// TIA Portal V20 export
// export: Created 2025-12-01T14:57:39.3017636Z, ExportSetting None, DisplayName Totally Integrated Automation Portal, DisplayVersion V20 Update 3, DisplayName TIA Portal Openness, DisplayVersion V20 Update 3, DisplayName TIA Portal Version Control Interface, DisplayVersion V20 Update 3, DisplayName STEP 7 Professional, DisplayVersion V20 Update 3, DisplayName STEP 7 Safety, DisplayVersion V20 Update 2, DisplayName WinCC Basic/Comfort/Advanced, DisplayVersion V20 Update 3, DisplayName WinCC Professional, DisplayVersion V20 Update 3, DisplayName WinCC Unified, DisplayVersion V20 Update 3
FUNCTION_BLOCK "FB370_ApiladorDeCajasPlastico"   // FB370, LAD
TITLE = Apilador de Cajas de Plastico
{ S7_Optimized_Access := 'FALSE' }
AUTHOR : MAQUINA
NAME : 20160211
VERSION : 3.2
// Dani Palacios: Modificación octubre 2017 para poder desabilitar la maquina con un bit (por ejemplo en la puesta a punto si no esta montada o en el simulador)
// La modificación esta sin probar y es todo lo relativo a la variable Maquina_Desabilitada
// (bloqueo evolución desde etapa 0, bloqueo activación salidas en etapa 0 , fin vi sin mirar detectores y activación posición de reposo sin mirar detectores y variabkles de fin de movimiento).
// ES RESPONSABILIDAD DEL QUE DESABILITA LA MAQUINA QUE ESTA ESTE EN UNA POSICION QUE PERMITA EL MOVIMIENTO DE LAS CARGAS A TRAVES DE ELLA
// stored: AutoNumber false, SetENOAutomatically false
   VAR_INPUT
      Maquina : UInt;   // Numero de Maquina (Mesa)
      Error_Tx : Bool;   // Error en el Tx
      EnTension : Bool;   // Existe Tension en la Mesa
      NodoNoPresente : Bool;   // Nodo No Presente >>> Var. LENZE de Elevacion
      ByteInicial : Int;   // Byte Inicial >>> Var. LENZE de Elevacion
      MAQx_DesHabilitada : Bool;   // Config MAQ. >>> DesHabilitada
      MAQx_SinPrimerCentrado : Bool;   // Config MAQ. >>> No Activar Primer Centrado (Antes de Entrada)
      MAQx_ActivarEspera : Bool;   // Config MAQ. >>> Sin Espera en Etapas
      MAQx_SinTopes : Bool;   // Config MAQ. >>> Sin Utilizar Topes (Los Centradores)
      TermicoFreno_ELEV : Bool;   // Termico del Freno de la Elevacion
      pHsMx_PresCarga : Bool;   // pHs de Presencia de Carga en la Maquina
      pHsMx_1 : Bool;   // pHs de la Mesa - Pos 1 de Av
      pHsMx_2 : Bool;   // pHs de la Mesa - Pos 2 de Av
      pHsMx_CtrEntrada : Bool;   // pHs Control de Entrada de Seguridad
      pHs_Referencia : Bool;   // pHs de Referencia >>> Var. LENZE de Elevacion
      EM_Up : Bool;   // Emergencia Arriba >>> Var. LENZE de Elevacion
      EM_Down : Bool;   // Emergencia Abajo >>> Var. LENZE de Elevacion
      CF1CF2_Cerrado : Bool;   // Centradores 1 y 2 Cerrados
      CF3CF4_Cerrado : Bool;   // Centradores 3 y 4 Cerrados
      CF5CF6_Cerrado : Bool;   // Centradores 5 y 6 Cerrados
      CF1CF2_Abierto : Bool;   // Centradores 1 y 2 Abiertos
      CF3CF4_Abierto : Bool;   // Centradores 3 y 4 Abiertos
      CF5CF6_Abierto : Bool;   // Centradores 5 y 6 Abiertos
      CM1CM2_Cerrado : Bool;   // Garras 1 y 2 Cerradas
      CM3CM4_Cerrado : Bool;   // Garras 3 y 4 Cerradas
      CM5CM6_Cerrado : Bool;   // Garras 5 y 6 Cerradas
      CM7CM8_Cerrado : Bool;   // Garras 7 y 8 Cerradas
      CM9CM10_Cerrado : Bool;   // Garras 9 y 10 Cerradas
      CM1CM2_Abierto : Bool;   // Garras 1 y 2 Abiertas
      CM3CM4_Abierto : Bool;   // Garras 3 y 4 Abiertas
      CM5CM6_Abierto : Bool;   // Garras 5 y 6 Abiertas
      CM7CM8_Abierto : Bool;   // Garras 7 y 8 Abiertas
      CM9CM10_Abierto : Bool;   // Garras 9 y 10 Abiertas
      GF1GF2_Cerrado : Bool;   // Guias superiores 1 y 2 Cerradas
      GF3GF4_Cerrado : Bool;   // Guias superiores 3 y 4 Cerradas
      GF1GF2_Abierto : Bool;   // Guias superiores 1 y 2 Abiertas
      GF3GF4_Abierto : Bool;   // Guias superiores 3 y 4 Abiertas
      EnMov_Centradores : Bool;   // Centradores >>> En Movimiento
      EnMov_Garras : Bool;   // Garras >>> En Movimiento
      EnMov_Guias : Bool;   // Guias >>> En Movimiento
      EnMov_Topes : Bool;   // Topes >>> En Movimiento
      SubirManual : Bool;   // Subir en Manual >>> Var. LENZE de Elevacion
      BajarManual : Bool;   // Bajar en Manual >>> Var. LENZE de Elevacion
      AutoManual : Bool;   // Posicionar en Manual (Para realizar Test de Posicion)
      Homing : Bool;   // Homing >>> Var. LENZE de Elevacion
      CajaGrande_EnEntrada : Bool;   // Caja Grande en Entrada >>> Interlock Mesa
      Apilador_AvisoEntrada : Bool;   // Aviso Entrada >>> Interlock Mesa
      Apilador_FinEntrada : Bool;   // FIn Entrada >>> Interlock Mesa
      ActivarGuias : Bool;   // Activar las Guias Superiores (Por altura de la Pila)
      V_TOut_MovVertical : Int := 15000;   // TimeOut del Movimiento Vertical
      V_TOut_Centradores : Int := 5000;   // TimeOut de los Centradores
      V_TOut_Garras : Int := 5000;   // TimeOut de las Garras
      V_TOut_Guias : Int := 5000;   // TimeOut de las Guias Superiores
      V_TOut_Topes : Int := 5000;   // TimeOut de los Topes
   END_VAR
   VAR_OUTPUT
      Apilador_EnReposo : Bool;   // En Reposo >>> Interlock Maquina
      Apialdor_PermisoEntrada : Bool;   // Permiso deEntrada >>> Interlock Maquina
   END_VAR
   VAR
      PosicionActual : Int;   // Var. LENZE de Elevacion >>> Posicion Actual
      ErrorSubjet : Word;   // Var LENZE de Elevacion
      ErrorID : Word;   // Var LENZE de Elevacion
      PosicionManual : UInt;   // Posicion para el Test Manual
      PosicionInicial : UInt;   // TRACKING >>> Posicion Inicial de la Orden de DesApilar Cajas
      PosicionFinal : UInt;   // TRACKING >>> Posicion Final de la Orden de DesApilar Cajas
      PosicionPreviaInicial : UInt;   // TRACKING >>> Posicion Previa a la inicial - Adelanto de Movimiento
      TipoAmarre : UInt;   // TRACKING >>> Tipo de Amarre de las Garras de la Orden de DesApilar Cajas
      OrdenApilar : Bool;   // TRACKING >>> Orden de DesApilar Cajas
      Fin_OrdenApilar : Bool;   // TRACKING >>> Fin de la Orden de DesApilar Cajas
      Caja_TipoEuroPool : Bool;   // TRACKING >>> Caja de tipo EuroPool
      Caja_DosPequenas : Bool;   // TRACKING >>> La Fila es de Dos Cajas Pequeñas
      Caja_UnaPequena : Bool;   // TRACKING >>> La Fila es de Una Caja Pequeña
      Caja_Grande : Bool;   // TRACKING >>> La Fila es de Una Caja Grande
      Reset_ET00 : Bool;
      Reset_ET01 : Bool;
      Apil_ET00 : Bool;
      Apil_ET01 : Bool;
      Apil_ET02 : Bool;
      Apil_ET03 : Bool;
      Apil_ET04 : Bool;
      Apil_ET05 : Bool;
      Apil_ET06 : Bool;
      Apil_ET07 : Bool;
      Apil_ET08 : Bool;
      Apil_ET09 : Bool;
      Apil_ET10 : Bool;
      Apil_ET11 : Bool;
      Apil_ET12 : Bool;
      Apil_ET13 : Bool;
      Apil_ET14 : Bool;
      Apil_ET15 : Bool;
      PosicionIntermedia : UInt;
      Posicion_OrdenMover : UInt;   // AUXILIAR >>> Posicion de la Orden a Mover el Elevacion
      OrdenMover : Bool;   // AUXILIAR >>> Orden de Mover el Elevacion
      Fin_OrdenMover : Bool;   // AUXILIAR >>> Orden de Mover el Elevacion
      MemoPosicionOK : Bool;   // AUXILIAR >>> Memoria de Posicion OK
      Carga_PosicionInicial : Bool;   // CARGA >>> Posicion Incial del Apilado de Cajas
      Carga_PosicionIntermedia : Bool;   // CARGA >>> Posicion Intermedia del Apilado de Cajas
      Carga_PosicionFinal : Bool;   // CARGA >>> Posicion Final del Apilado de Cajas
      Carga_PosicionPreviaIncial : Bool;   // CARGA >>> Posicion Previa Inicial del Apilado de Cajas
      Carga_PosicionManual : Bool;   // CARGA >>> Posicion Manual de la Orden de Test
      ErrorVariador : Bool;   // AUXILIAR >>> Error del Variador
      ReferenciaOK : Bool;   // AUXILIAR >>> Referencia OK del Variador
      MemoHomingAuto : Bool;   // AUXILIAR >>> Memoria del Homing Automatico del Variador
      TIM_EsperaMover { S7_SetPoint := 'True'} : TON_TIME;   // TIM de Espera de Activar Orden al Var de LENZE (200ms)
      TIM_EsperaET02 { S7_SetPoint := 'True'} : TON_TIME;   // TIM de Espera para Activar ET02 (100ms)
      TIM_EsperaET05 { S7_SetPoint := 'True'} : TON_TIME;   // TIM de Espera para Activar ET05 (100ms)
      TIM_EsperaET13 { S7_SetPoint := 'True'} : TON_TIME;   // TIM de Espera para Activar ET13 (100ms)
      TMP_EnTension { S7_SetPoint := 'True'} : "FB910_CNT_UHS";
      TOut_MovVertical { S7_SetPoint := 'True'} : "FB910_CNT_UHS";   // TimeOut del Movimiento Vertical
      TOut_Centradores { S7_SetPoint := 'True'} : "FB910_CNT_UHS";   // TimeOut de los Centradores
      TOut_Garras { S7_SetPoint := 'True'} : "FB910_CNT_UHS";   // TimeOut de las Garras
      TOut_Guias { S7_SetPoint := 'True'} : "FB910_CNT_UHS";   // TimeOut de las Guias Superiores
      TOut_Topes { S7_SetPoint := 'True'} : "FB910_CNT_UHS";   // TimeOut de los Topes
      MA_Cerrar_CF1CF2 : Bool;   // ????
      MA_Cerrar_CF3CF4 : Bool;   // ????
      MA_Cerrar_CF5CF6 : Bool;   // ????
      MA_Abrir_CF1CF2 : Bool;   // ????
      MA_Abrir_CF3CF4 : Bool;   // ????
      MA_Abrir_CF5CF6 { ExternalVisible := 'False'} : Bool;   // ????
      MA_Cerrar_CM1CM2 : Bool;   // ????
      MA_Cerrar_CM3CM4 : Bool;   // ????
      MA_Cerrar_CM5CM6 : Bool;   // ????
      MA_Cerrar_CM7CM8 : Bool;   // ????
      MA_Cerrar_CM9CM10 : Bool;   // ????
      MA_Abrir_CM1CM2 : Bool;   // ????
      MA_Abrir_CM3CM4 : Bool;   // ????
      MA_Abrir_CM5CM6 : Bool;   // ????
      MA_Abrir_CM7CM8 : Bool;   // ????
      MA_Abrir_CM9CM10 : Bool;   // ????
      MA_Cerrar_GF1GF2 : Bool;   // ????
      MA_Cerrar_GF3GF4 : Bool;   // ????
      MA_Abrir_GF1GF2 : Bool;   // ????
      MA_Abrir_GF3GF4 : Bool;   // ????
   END_VAR
   VAR_TEMP
      EstadoZona : "EstadoZona";   // Estado de Zona de la Mesa
      EstadoMAQ : "EstadoMaquina_ApiladorDeCajasPlastico";   // Estado del Vehiculo Inteliguente de la Maquina
      MAQx_AutoHoming : Bool;   // Config >>> Var. LENZE con Auto Homing
      MAQx_EncoderIncremental : Bool;   // Config >>> Var. LENZE con Encoder Incremental
      MAQx_ActivarAutoManual : Bool;   // Config >>> Activacion para el Test de posicionamiento manual
      MAQx_SinAbrirTopes : Bool;   // Config MAQ. >>> No Abrir Topes - Despues de Entrada
      MAQx_EntradaSinEspera : Bool;   // Config MAQ. >>> No Esperar el Cerrar Topes - Inicio de Entrada
      CentradoresCerrados : Bool;   // AUXILIAR >>> Cerrados los Centradores
      CentradoresAbiertos : Bool;   // AUXILIAR >>> Abiertos los Centradores
      TopesCerrados : Bool;   // AUXILIAR >>> Cerrados los Topes
      GarrasCerradas : Bool;   // AUXILIAR >>> Cerradas las Garras
      GarrasAbiertas : Bool;   // AUXILIAR >>> Abiertas las Garras
      GuiasCerradas : Bool;   // AUXILIAR >>> Cerradas las Guias Superiores
      GuiasAbiertas : Bool;   // AUXILIAR >>> Abiertas las Guias Superiores
      MA_CerrarCentradores : Bool;   // AUXILIAR >>> Cerrar los Centradores
      MA_AbrirCentradores : Bool;   // AUXILIAR >>> Abrir los Centradores
      MA_CerrarTopes : Bool;   // AUXILIAR >>> Cerrar los Topes
      MA_CerrarGarras : Bool;   // AUXILIAR >>> Cerrar las Garras
      MA_AbrirGarras : Bool;   // AUXILIAR >>> Abrir las Garras
      MA_CerrarGuias : Bool;   // AUXILIAR >>> Cerrar las Guias Superiores
      MA_AbrirGuias : Bool;   // AUXILIAR >>> Abrir las Guias Superiores
      Aux_ET00 : Bool;
   END_VAR
BEGIN

REGION Network 1: Configuraciones Especiales - Config >>> Var. LENZE de Elevacion
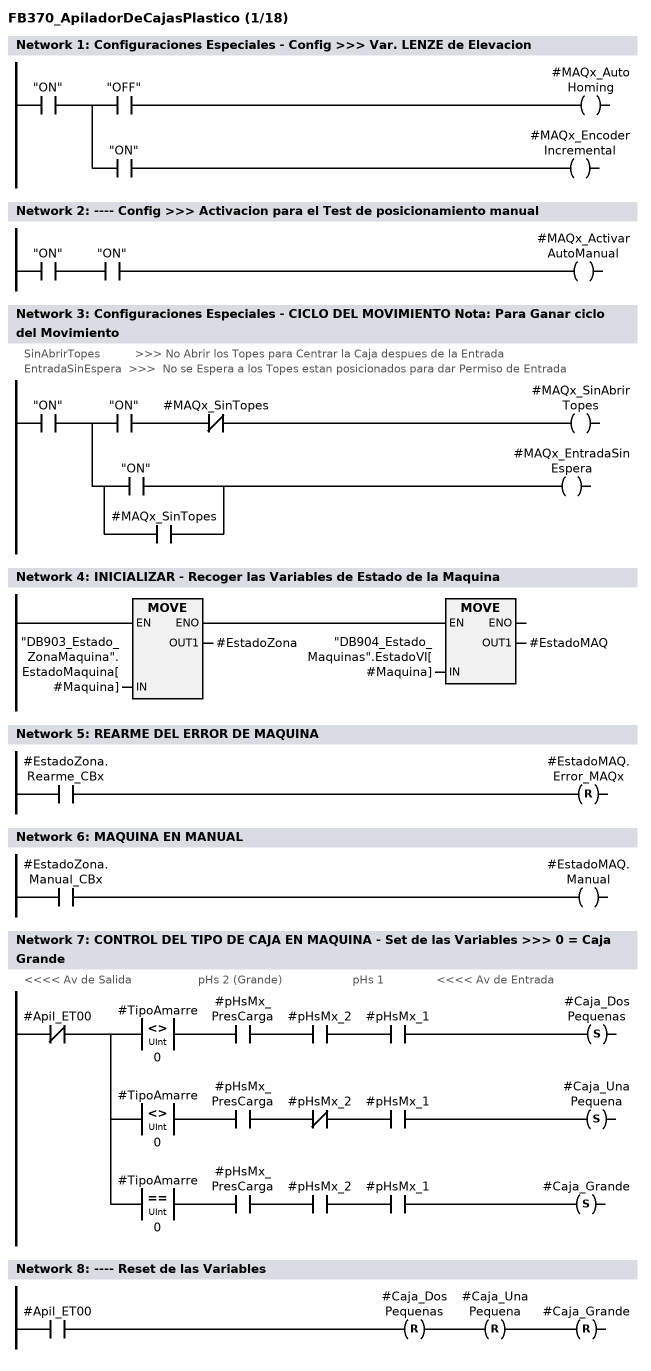
   RUNG wire#powerrail
      Contact( "ON" )
      wire#w1
      Contact( "OFF" )
      Coil( #MAQx_AutoHoming )
   END_RUNG
   RUNG wire#w1
      Contact( "ON" )
      Coil( #MAQx_EncoderIncremental )
   END_RUNG
   // the same network as SCL:
   #MAQx_AutoHoming := "ON" AND "OFF";
   #MAQx_EncoderIncremental := "ON" AND "ON";
END_REGION

REGION Network 2: ---- Config >>> Activacion para el Test de posicionamiento manual
   RUNG wire#powerrail
      Contact( "ON" )
      Contact( "ON" )
      Coil( #MAQx_ActivarAutoManual )
   END_RUNG
   // the same network as SCL:
   #MAQx_ActivarAutoManual := "ON" AND "ON";
END_REGION

REGION Network 3: Configuraciones Especiales - CICLO DEL MOVIMIENTO Nota: Para Ganar ciclo del Movimiento
   // SinAbrirTopes          >>> No Abrir los Topes para Centrar la Caja despues de la Entrada
   // EntradaSinEspera  >>>  No se Espera a los Topes estan posicionados para dar Permiso de Entrada
   RUNG wire#powerrail
      Contact( "ON" )
      wire#w1
      Contact( "ON" )
      I_Contact( #MAQx_SinTopes )
      Coil( #MAQx_SinAbrirTopes )
   END_RUNG
   RUNG wire#w1
      Contact( "ON" )
      wire#w2
      Coil( #MAQx_EntradaSinEspera )
   END_RUNG
   RUNG wire#w1
      Contact( #MAQx_SinTopes )
   END_RUNG wire#w2
   // the same network as SCL:
   #MAQx_SinAbrirTopes := "ON" AND "ON" AND NOT #MAQx_SinTopes;
   #MAQx_EntradaSinEspera := "ON" AND ("ON" OR #MAQx_SinTopes);
END_REGION

REGION Network 4: INICIALIZAR - Recoger las Variables de Estado de la Maquina
   RUNG wire#powerrail
      Move(in := "DB903_Estado_ZonaMaquina".EstadoMaquina[#Maquina], out1 => #EstadoZona)
      Move(in := "DB904_Estado_Maquinas".EstadoVI[#Maquina], out1 => #EstadoMAQ)
   END_RUNG
   // the same network as SCL:
   #EstadoZona := "DB903_Estado_ZonaMaquina".EstadoMaquina[#Maquina];
   #EstadoMAQ := "DB904_Estado_Maquinas".EstadoVI[#Maquina];
END_REGION

REGION Network 5: REARME DEL ERROR DE MAQUINA
   RUNG wire#powerrail
      Contact( #EstadoZona.Rearme_CBx )
      R_Coil( #EstadoMAQ.Error_MAQx )
   END_RUNG
   // the same network as SCL:
   IF #EstadoZona.Rearme_CBx THEN #EstadoMAQ.Error_MAQx := FALSE; END_IF;
END_REGION

REGION Network 6: MAQUINA EN MANUAL
   RUNG wire#powerrail
      Contact( #EstadoZona.Manual_CBx )
      Coil( #EstadoMAQ.Manual )
   END_RUNG
   // the same network as SCL:
   #EstadoMAQ.Manual := #EstadoZona.Manual_CBx;
END_REGION

REGION Network 7: CONTROL DEL TIPO DE CAJA EN MAQUINA - Set de las Variables >>> 0 = Caja Grande
   // <<<< Av de Salida                   pHs 2 (Grande)                    pHs 1               <<<< Av de Entrada
   RUNG wire#powerrail
      I_Contact( #Apil_ET00 )
      wire#w1
      { S7_Templates := "SrcType := UInt" } NE_Contact(in1 := #TipoAmarre, in2 := 0)
      Contact( #pHsMx_PresCarga )
      Contact( #pHsMx_2 )
      Contact( #pHsMx_1 )
      S_Coil( #Caja_DosPequenas )
   END_RUNG
   RUNG wire#w1
      { S7_Templates := "SrcType := UInt" } NE_Contact(in1 := #TipoAmarre, in2 := 0)
      Contact( #pHsMx_PresCarga )
      I_Contact( #pHsMx_2 )
      Contact( #pHsMx_1 )
      S_Coil( #Caja_UnaPequena )
   END_RUNG
   RUNG wire#w1
      { S7_Templates := "SrcType := UInt" } EQ_Contact(in1 := #TipoAmarre, in2 := 0)
      Contact( #pHsMx_PresCarga )
      Contact( #pHsMx_2 )
      Contact( #pHsMx_1 )
      S_Coil( #Caja_Grande )
   END_RUNG
   // the same network as SCL:
   IF NOT #Apil_ET00 AND (#TipoAmarre <> 0) AND #pHsMx_PresCarga AND #pHsMx_2 AND #pHsMx_1 THEN
       #Caja_DosPequenas := TRUE;
   END_IF;
   IF NOT #Apil_ET00 AND (#TipoAmarre <> 0) AND #pHsMx_PresCarga AND NOT #pHsMx_2 AND #pHsMx_1 THEN
       #Caja_UnaPequena := TRUE;
   END_IF;
   IF NOT #Apil_ET00 AND (#TipoAmarre = 0) AND #pHsMx_PresCarga AND #pHsMx_2 AND #pHsMx_1 THEN
       #Caja_Grande := TRUE;
   END_IF;
END_REGION

REGION Network 8: ---- Reset de las Variables
   RUNG wire#powerrail
      Contact( #Apil_ET00 )
      R_Coil( #Caja_DosPequenas )
      R_Coil( #Caja_UnaPequena )
      R_Coil( #Caja_Grande )
   END_RUNG
   // the same network as SCL:
   IF #Apil_ET00 THEN
       #Caja_DosPequenas := FALSE;
       #Caja_UnaPequena := FALSE;
       #Caja_Grande := FALSE;
   END_IF;
END_REGION

REGION Network 9: ---- Config >>> Caja de tipo EuroPool
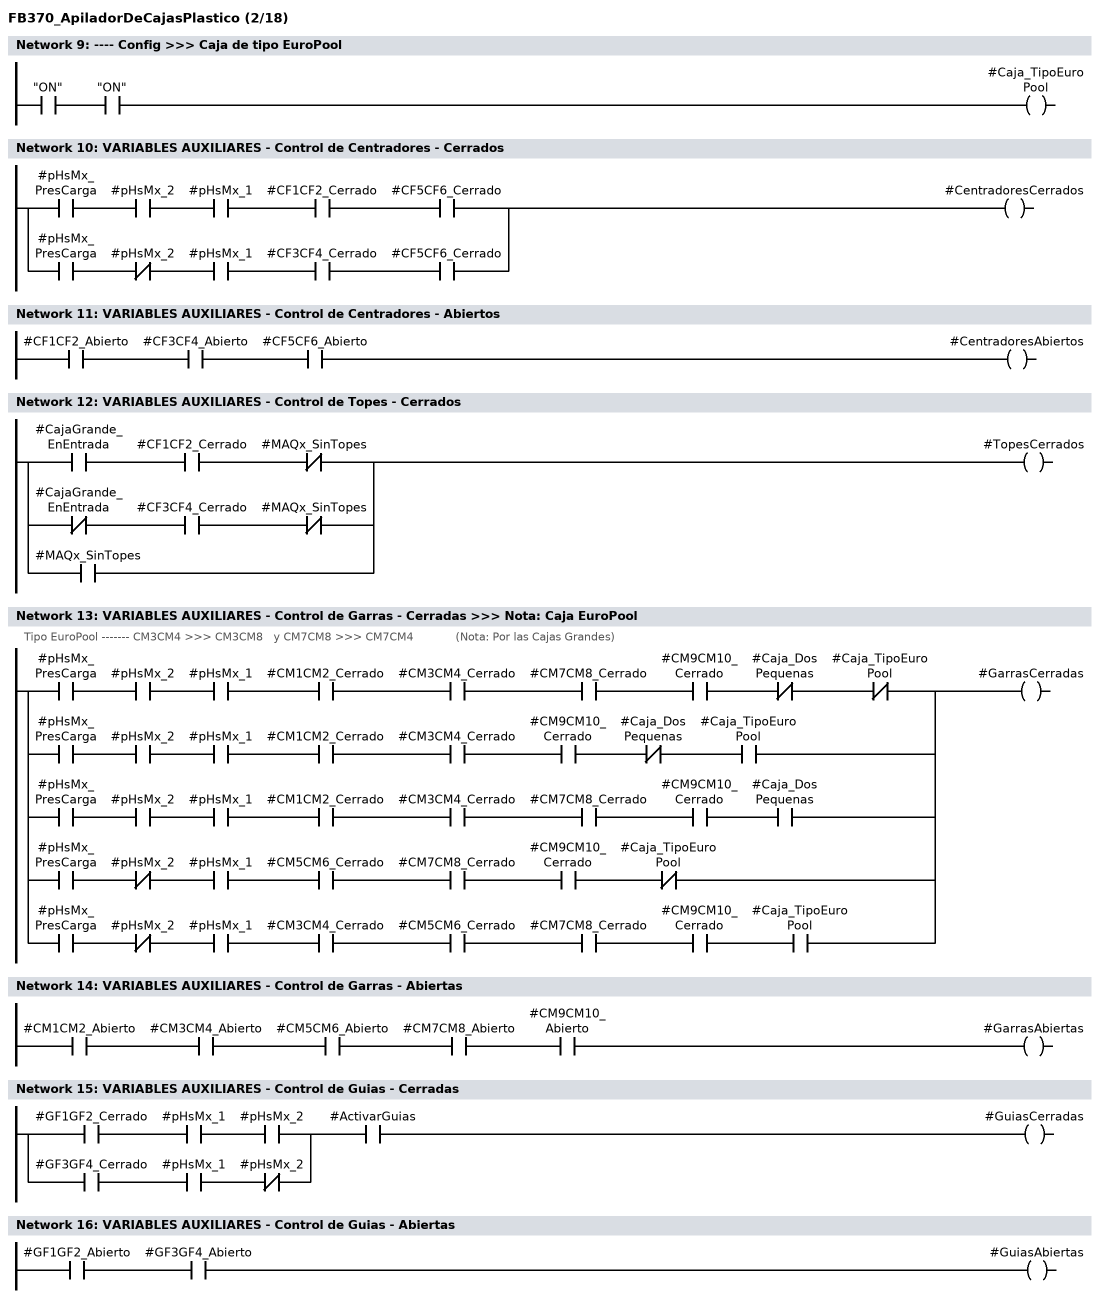
   RUNG wire#powerrail
      Contact( "ON" )
      Contact( "ON" )
      Coil( #Caja_TipoEuroPool )
   END_RUNG
   // the same network as SCL:
   #Caja_TipoEuroPool := "ON" AND "ON";
END_REGION

REGION Network 10: VARIABLES AUXILIARES - Control de Centradores - Cerrados
   RUNG wire#powerrail
      Contact( #pHsMx_PresCarga )
      Contact( #pHsMx_2 )
      Contact( #pHsMx_1 )
      Contact( #CF1CF2_Cerrado )
      Contact( #CF5CF6_Cerrado )
      wire#w1
      Coil( #CentradoresCerrados )
   END_RUNG
   RUNG wire#powerrail
      Contact( #pHsMx_PresCarga )
      I_Contact( #pHsMx_2 )
      Contact( #pHsMx_1 )
      Contact( #CF3CF4_Cerrado )
      Contact( #CF5CF6_Cerrado )
   END_RUNG wire#w1
   // the same network as SCL:
   #CentradoresCerrados := (#pHsMx_PresCarga AND #pHsMx_2 AND #pHsMx_1 AND #CF1CF2_Cerrado AND #CF5CF6_Cerrado) OR (#pHsMx_PresCarga AND NOT #pHsMx_2 AND #pHsMx_1 AND #CF3CF4_Cerrado AND #CF5CF6_Cerrado);
END_REGION

REGION Network 11: VARIABLES AUXILIARES - Control de Centradores - Abiertos
   RUNG wire#powerrail
      Contact( #CF1CF2_Abierto )
      Contact( #CF3CF4_Abierto )
      Contact( #CF5CF6_Abierto )
      Coil( #CentradoresAbiertos )
   END_RUNG
   // the same network as SCL:
   #CentradoresAbiertos := #CF1CF2_Abierto AND #CF3CF4_Abierto AND #CF5CF6_Abierto;
END_REGION

REGION Network 12: VARIABLES AUXILIARES - Control de Topes - Cerrados
   RUNG wire#powerrail
      Contact( #CajaGrande_EnEntrada )
      Contact( #CF1CF2_Cerrado )
      I_Contact( #MAQx_SinTopes )
      wire#w1
      Coil( #TopesCerrados )
   END_RUNG
   RUNG wire#powerrail
      I_Contact( #CajaGrande_EnEntrada )
      Contact( #CF3CF4_Cerrado )
      I_Contact( #MAQx_SinTopes )
   END_RUNG wire#w1
   RUNG wire#powerrail
      Contact( #MAQx_SinTopes )
   END_RUNG wire#w1
   // the same network as SCL:
   #TopesCerrados := (#CajaGrande_EnEntrada AND #CF1CF2_Cerrado AND NOT #MAQx_SinTopes) OR (NOT #CajaGrande_EnEntrada AND #CF3CF4_Cerrado AND NOT #MAQx_SinTopes) OR #MAQx_SinTopes;
END_REGION

REGION Network 13: VARIABLES AUXILIARES - Control de Garras - Cerradas >>> Nota: Caja EuroPool
   // Tipo EuroPool ------- CM3CM4 >>> CM3CM8   y CM7CM8 >>> CM7CM4            (Nota: Por las Cajas Grandes)
   RUNG wire#powerrail
      Contact( #pHsMx_PresCarga )
      Contact( #pHsMx_2 )
      Contact( #pHsMx_1 )
      Contact( #CM1CM2_Cerrado )
      Contact( #CM3CM4_Cerrado )
      Contact( #CM7CM8_Cerrado )
      Contact( #CM9CM10_Cerrado )
      I_Contact( #Caja_DosPequenas )
      I_Contact( #Caja_TipoEuroPool )
      wire#w1
      Coil( #GarrasCerradas )
   END_RUNG
   RUNG wire#powerrail
      Contact( #pHsMx_PresCarga )
      Contact( #pHsMx_2 )
      Contact( #pHsMx_1 )
      Contact( #CM1CM2_Cerrado )
      Contact( #CM3CM4_Cerrado )
      Contact( #CM9CM10_Cerrado )
      I_Contact( #Caja_DosPequenas )
      Contact( #Caja_TipoEuroPool )
   END_RUNG wire#w1
   RUNG wire#powerrail
      Contact( #pHsMx_PresCarga )
      Contact( #pHsMx_2 )
      Contact( #pHsMx_1 )
      Contact( #CM1CM2_Cerrado )
      Contact( #CM3CM4_Cerrado )
      Contact( #CM7CM8_Cerrado )
      Contact( #CM9CM10_Cerrado )
      Contact( #Caja_DosPequenas )
   END_RUNG wire#w1
   RUNG wire#powerrail
      Contact( #pHsMx_PresCarga )
      I_Contact( #pHsMx_2 )
      Contact( #pHsMx_1 )
      Contact( #CM5CM6_Cerrado )
      Contact( #CM7CM8_Cerrado )
      Contact( #CM9CM10_Cerrado )
      I_Contact( #Caja_TipoEuroPool )
   END_RUNG wire#w1
   RUNG wire#powerrail
      Contact( #pHsMx_PresCarga )
      I_Contact( #pHsMx_2 )
      Contact( #pHsMx_1 )
      Contact( #CM3CM4_Cerrado )
      Contact( #CM5CM6_Cerrado )
      Contact( #CM7CM8_Cerrado )
      Contact( #CM9CM10_Cerrado )
      Contact( #Caja_TipoEuroPool )
   END_RUNG wire#w1
   // the same network as SCL:
   #GarrasCerradas := (#pHsMx_PresCarga AND #pHsMx_2 AND #pHsMx_1 AND #CM1CM2_Cerrado AND #CM3CM4_Cerrado AND #CM7CM8_Cerrado AND #CM9CM10_Cerrado AND NOT #Caja_DosPequenas AND NOT #Caja_TipoEuroPool) OR (#pHsMx_PresCarga AND #pHsMx_2 AND #pHsMx_1 AND #CM1CM2_Cerrado AND #CM3CM4_Cerrado AND #CM9CM10_Cerrado AND NOT #Caja_DosPequenas AND #Caja_TipoEuroPool) OR (#pHsMx_PresCarga AND #pHsMx_2 AND #pHsMx_1 AND #CM1CM2_Cerrado AND #CM3CM4_Cerrado AND #CM7CM8_Cerrado AND #CM9CM10_Cerrado AND #Caja_DosPequenas) OR (#pHsMx_PresCarga AND NOT #pHsMx_2 AND #pHsMx_1 AND #CM5CM6_Cerrado AND #CM7CM8_Cerrado AND #CM9CM10_Cerrado AND NOT #Caja_TipoEuroPool) OR (#pHsMx_PresCarga AND NOT #pHsMx_2 AND #pHsMx_1 AND #CM3CM4_Cerrado AND #CM5CM6_Cerrado AND #CM7CM8_Cerrado AND #CM9CM10_Cerrado AND #Caja_TipoEuroPool);
END_REGION

REGION Network 14: VARIABLES AUXILIARES - Control de Garras - Abiertas
   RUNG wire#powerrail
      Contact( #CM1CM2_Abierto )
      Contact( #CM3CM4_Abierto )
      Contact( #CM5CM6_Abierto )
      Contact( #CM7CM8_Abierto )
      Contact( #CM9CM10_Abierto )
      Coil( #GarrasAbiertas )
   END_RUNG
   // the same network as SCL:
   #GarrasAbiertas := #CM1CM2_Abierto AND #CM3CM4_Abierto AND #CM5CM6_Abierto AND #CM7CM8_Abierto AND #CM9CM10_Abierto;
END_REGION

REGION Network 15: VARIABLES AUXILIARES - Control de Guias - Cerradas
   RUNG wire#powerrail
      Contact( #GF1GF2_Cerrado )
      Contact( #pHsMx_1 )
      Contact( #pHsMx_2 )
      wire#w1
      Contact( #ActivarGuias )
      Coil( #GuiasCerradas )
   END_RUNG
   RUNG wire#powerrail
      Contact( #GF3GF4_Cerrado )
      Contact( #pHsMx_1 )
      I_Contact( #pHsMx_2 )
   END_RUNG wire#w1
   // the same network as SCL:
   #GuiasCerradas := ((#GF1GF2_Cerrado AND #pHsMx_1 AND #pHsMx_2) OR (#GF3GF4_Cerrado AND #pHsMx_1 AND NOT #pHsMx_2)) AND #ActivarGuias;
END_REGION

REGION Network 16: VARIABLES AUXILIARES - Control de Guias - Abiertas
   RUNG wire#powerrail
      Contact( #GF1GF2_Abierto )
      Contact( #GF3GF4_Abierto )
      Coil( #GuiasAbiertas )
   END_RUNG
   // the same network as SCL:
   #GuiasAbiertas := #GF1GF2_Abierto AND #GF3GF4_Abierto;
END_REGION

REGION Network 17: VARIADOR LENZE - MEMORIA del Fin del Movimiento
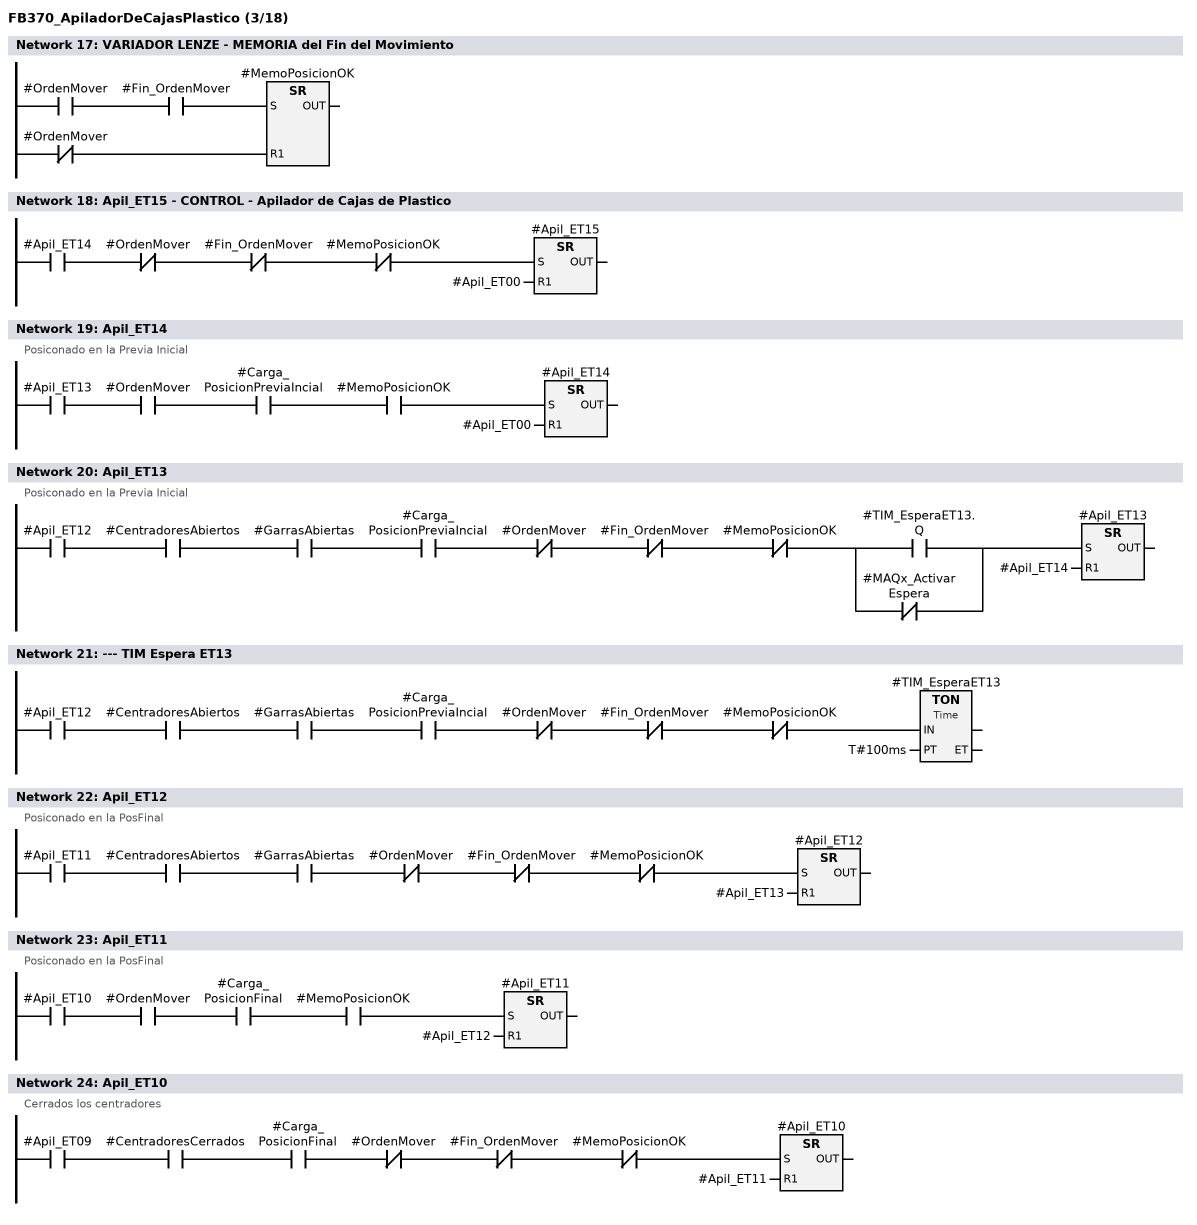
   RUNG wire#powerrail
      Contact( #OrdenMover )
      Contact( #Fin_OrdenMover )
      S_SR(operand := #MemoPosicionOK, r1 := wire#w1)
   END_RUNG
   RUNG wire#powerrail
      I_Contact( #OrdenMover )
   END_RUNG wire#w1
   // the same network as SCL:
   IF #OrdenMover AND #Fin_OrdenMover THEN
       #MemoPosicionOK := TRUE;   // SR flip-flop
   END_IF;
   IF NOT #OrdenMover THEN #MemoPosicionOK := FALSE; END_IF;
END_REGION

REGION Network 18: Apil_ET15 - CONTROL - Apilador de Cajas de Plastico
   RUNG wire#powerrail
      Contact( #Apil_ET14 )
      I_Contact( #OrdenMover )
      I_Contact( #Fin_OrdenMover )
      I_Contact( #MemoPosicionOK )
      S_SR(operand := #Apil_ET15, r1 := #Apil_ET00)
   END_RUNG
   // the same network as SCL:
   IF #Apil_ET14 AND NOT #OrdenMover AND NOT #Fin_OrdenMover AND NOT #MemoPosicionOK THEN
       #Apil_ET15 := TRUE;   // SR flip-flop
   END_IF;
   IF #Apil_ET00 THEN #Apil_ET15 := FALSE; END_IF;
END_REGION

REGION Network 19: Apil_ET14
   // Posiconado en la Previa Inicial
   RUNG wire#powerrail
      Contact( #Apil_ET13 )
      Contact( #OrdenMover )
      Contact( #Carga_PosicionPreviaIncial )
      Contact( #MemoPosicionOK )
      S_SR(operand := #Apil_ET14, r1 := #Apil_ET00)
   END_RUNG
   // the same network as SCL:
   IF #Apil_ET13 AND #OrdenMover AND #Carga_PosicionPreviaIncial AND #MemoPosicionOK THEN
       #Apil_ET14 := TRUE;   // SR flip-flop
   END_IF;
   IF #Apil_ET00 THEN #Apil_ET14 := FALSE; END_IF;
END_REGION

REGION Network 20: Apil_ET13
   // Posiconado en la Previa Inicial
   RUNG wire#powerrail
      Contact( #Apil_ET12 )
      Contact( #CentradoresAbiertos )
      Contact( #GarrasAbiertas )
      Contact( #Carga_PosicionPreviaIncial )
      I_Contact( #OrdenMover )
      I_Contact( #Fin_OrdenMover )
      I_Contact( #MemoPosicionOK )
      wire#w1
      Contact( #TIM_EsperaET13.Q )
      wire#w2
      S_SR(operand := #Apil_ET13, r1 := #Apil_ET14)
   END_RUNG
   RUNG wire#w1
      I_Contact( #MAQx_ActivarEspera )
   END_RUNG wire#w2
   // the same network as SCL:
   IF #Apil_ET12 AND #CentradoresAbiertos AND #GarrasAbiertas AND #Carga_PosicionPreviaIncial AND NOT #OrdenMover AND NOT #Fin_OrdenMover AND NOT #MemoPosicionOK AND (#TIM_EsperaET13.Q OR NOT #MAQx_ActivarEspera) THEN
       #Apil_ET13 := TRUE;   // SR flip-flop
   END_IF;
   IF #Apil_ET14 THEN #Apil_ET13 := FALSE; END_IF;
END_REGION

REGION Network 21: --- TIM Espera ET13
   RUNG wire#powerrail
      Contact( #Apil_ET12 )
      Contact( #CentradoresAbiertos )
      Contact( #GarrasAbiertas )
      Contact( #Carga_PosicionPreviaIncial )
      I_Contact( #OrdenMover )
      I_Contact( #Fin_OrdenMover )
      I_Contact( #MemoPosicionOK )
      { S7_Templates := "time_type := Time" } #TIM_EsperaET13.TON(pt := T#100ms, et =>)
   END_RUNG
   // the same network as SCL:
   #TIM_EsperaET13(IN := #Apil_ET12 AND #CentradoresAbiertos AND #GarrasAbiertas AND #Carga_PosicionPreviaIncial AND NOT #OrdenMover AND NOT #Fin_OrdenMover AND NOT #MemoPosicionOK,   // TON
                   PT := T#100ms);
END_REGION

REGION Network 22: Apil_ET12
   // Posiconado en la PosFinal
   RUNG wire#powerrail
      Contact( #Apil_ET11 )
      Contact( #CentradoresAbiertos )
      Contact( #GarrasAbiertas )
      I_Contact( #OrdenMover )
      I_Contact( #Fin_OrdenMover )
      I_Contact( #MemoPosicionOK )
      S_SR(operand := #Apil_ET12, r1 := #Apil_ET13)
   END_RUNG
   // the same network as SCL:
   IF #Apil_ET11 AND #CentradoresAbiertos AND #GarrasAbiertas AND NOT #OrdenMover AND NOT #Fin_OrdenMover AND NOT #MemoPosicionOK THEN
       #Apil_ET12 := TRUE;   // SR flip-flop
   END_IF;
   IF #Apil_ET13 THEN #Apil_ET12 := FALSE; END_IF;
END_REGION

REGION Network 23: Apil_ET11
   // Posiconado en la PosFinal
   RUNG wire#powerrail
      Contact( #Apil_ET10 )
      Contact( #OrdenMover )
      Contact( #Carga_PosicionFinal )
      Contact( #MemoPosicionOK )
      S_SR(operand := #Apil_ET11, r1 := #Apil_ET12)
   END_RUNG
   // the same network as SCL:
   IF #Apil_ET10 AND #OrdenMover AND #Carga_PosicionFinal AND #MemoPosicionOK THEN
       #Apil_ET11 := TRUE;   // SR flip-flop
   END_IF;
   IF #Apil_ET12 THEN #Apil_ET11 := FALSE; END_IF;
END_REGION

REGION Network 24: Apil_ET10
   // Cerrados los centradores
   RUNG wire#powerrail
      Contact( #Apil_ET09 )
      Contact( #CentradoresCerrados )
      Contact( #Carga_PosicionFinal )
      I_Contact( #OrdenMover )
      I_Contact( #Fin_OrdenMover )
      I_Contact( #MemoPosicionOK )
      S_SR(operand := #Apil_ET10, r1 := #Apil_ET11)
   END_RUNG
   // the same network as SCL:
   IF #Apil_ET09 AND #CentradoresCerrados AND #Carga_PosicionFinal AND NOT #OrdenMover AND NOT #Fin_OrdenMover AND NOT #MemoPosicionOK THEN
       #Apil_ET10 := TRUE;   // SR flip-flop
   END_IF;
   IF #Apil_ET11 THEN #Apil_ET10 := FALSE; END_IF;
END_REGION

REGION Network 25: Apil_ET09
   // SinAbrirTopes          >>> No Abrir los Topes para Centrar la Caja despues de la Entrada
   // Abiertos los Centradores
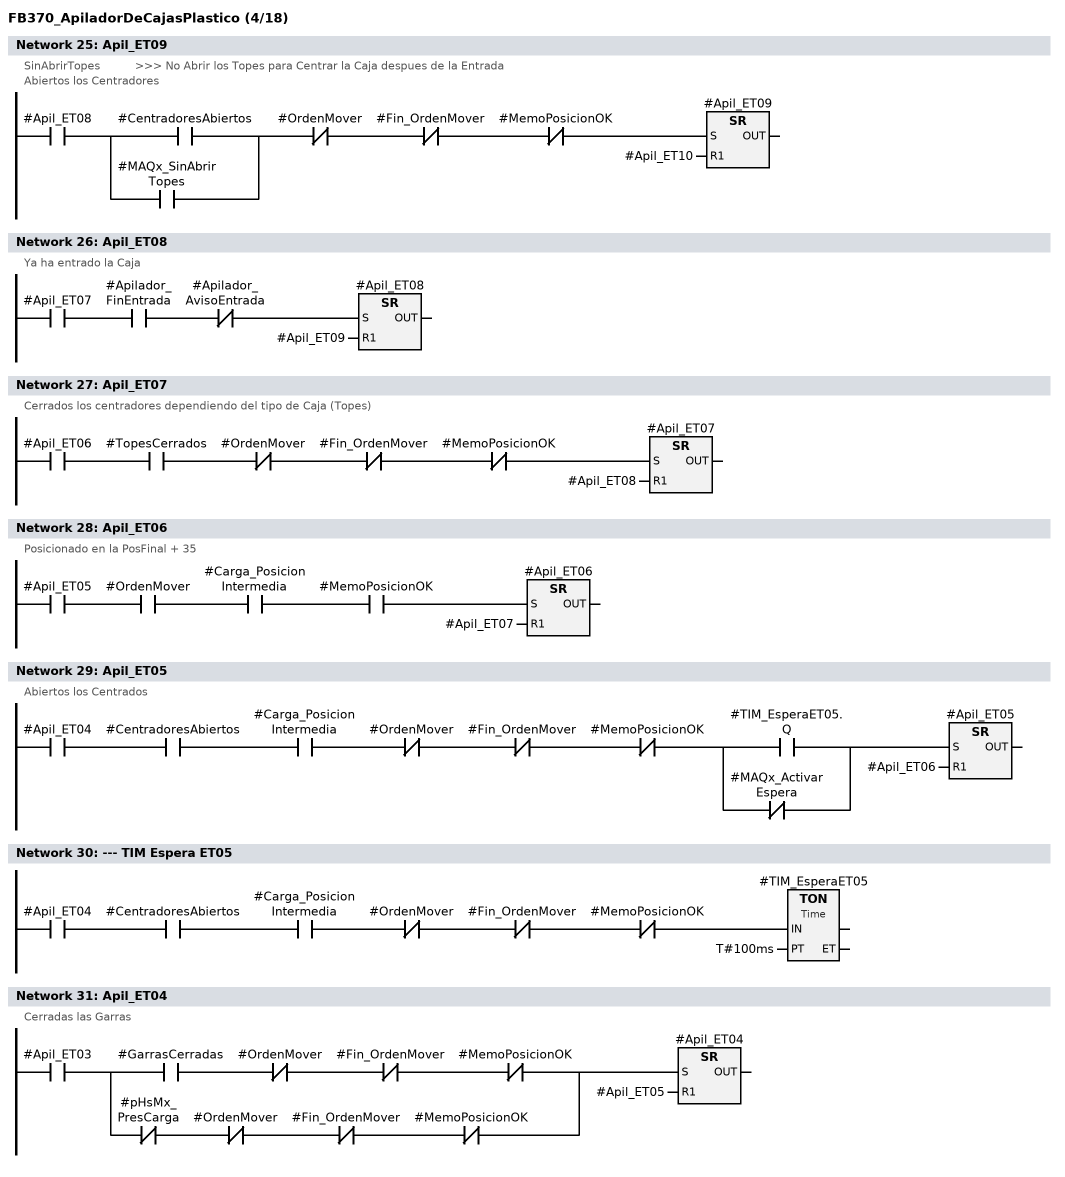
   RUNG wire#powerrail
      Contact( #Apil_ET08 )
      wire#w1
      Contact( #CentradoresAbiertos )
      wire#w2
      I_Contact( #OrdenMover )
      I_Contact( #Fin_OrdenMover )
      I_Contact( #MemoPosicionOK )
      S_SR(operand := #Apil_ET09, r1 := #Apil_ET10)
   END_RUNG
   RUNG wire#w1
      Contact( #MAQx_SinAbrirTopes )
   END_RUNG wire#w2
   // the same network as SCL:
   IF #Apil_ET08 AND (#CentradoresAbiertos OR #MAQx_SinAbrirTopes) AND NOT #OrdenMover AND NOT #Fin_OrdenMover AND NOT #MemoPosicionOK THEN
       #Apil_ET09 := TRUE;   // SR flip-flop
   END_IF;
   IF #Apil_ET10 THEN #Apil_ET09 := FALSE; END_IF;
END_REGION

REGION Network 26: Apil_ET08
   // Ya ha entrado la Caja
   RUNG wire#powerrail
      Contact( #Apil_ET07 )
      Contact( #Apilador_FinEntrada )
      I_Contact( #Apilador_AvisoEntrada )
      S_SR(operand := #Apil_ET08, r1 := #Apil_ET09)
   END_RUNG
   // the same network as SCL:
   IF #Apil_ET07 AND #Apilador_FinEntrada AND NOT #Apilador_AvisoEntrada THEN
       #Apil_ET08 := TRUE;   // SR flip-flop
   END_IF;
   IF #Apil_ET09 THEN #Apil_ET08 := FALSE; END_IF;
END_REGION

REGION Network 27: Apil_ET07
   // Cerrados los centradores dependiendo del tipo de Caja (Topes)
   RUNG wire#powerrail
      Contact( #Apil_ET06 )
      Contact( #TopesCerrados )
      I_Contact( #OrdenMover )
      I_Contact( #Fin_OrdenMover )
      I_Contact( #MemoPosicionOK )
      S_SR(operand := #Apil_ET07, r1 := #Apil_ET08)
   END_RUNG
   // the same network as SCL:
   IF #Apil_ET06 AND #TopesCerrados AND NOT #OrdenMover AND NOT #Fin_OrdenMover AND NOT #MemoPosicionOK THEN
       #Apil_ET07 := TRUE;   // SR flip-flop
   END_IF;
   IF #Apil_ET08 THEN #Apil_ET07 := FALSE; END_IF;
END_REGION

REGION Network 28: Apil_ET06
   // Posicionado en la PosFinal + 35
   RUNG wire#powerrail
      Contact( #Apil_ET05 )
      Contact( #OrdenMover )
      Contact( #Carga_PosicionIntermedia )
      Contact( #MemoPosicionOK )
      S_SR(operand := #Apil_ET06, r1 := #Apil_ET07)
   END_RUNG
   // the same network as SCL:
   IF #Apil_ET05 AND #OrdenMover AND #Carga_PosicionIntermedia AND #MemoPosicionOK THEN
       #Apil_ET06 := TRUE;   // SR flip-flop
   END_IF;
   IF #Apil_ET07 THEN #Apil_ET06 := FALSE; END_IF;
END_REGION

REGION Network 29: Apil_ET05
   // Abiertos los Centrados
   RUNG wire#powerrail
      Contact( #Apil_ET04 )
      Contact( #CentradoresAbiertos )
      Contact( #Carga_PosicionIntermedia )
      I_Contact( #OrdenMover )
      I_Contact( #Fin_OrdenMover )
      I_Contact( #MemoPosicionOK )
      wire#w1
      Contact( #TIM_EsperaET05.Q )
      wire#w2
      S_SR(operand := #Apil_ET05, r1 := #Apil_ET06)
   END_RUNG
   RUNG wire#w1
      I_Contact( #MAQx_ActivarEspera )
   END_RUNG wire#w2
   // the same network as SCL:
   IF #Apil_ET04 AND #CentradoresAbiertos AND #Carga_PosicionIntermedia AND NOT #OrdenMover AND NOT #Fin_OrdenMover AND NOT #MemoPosicionOK AND (#TIM_EsperaET05.Q OR NOT #MAQx_ActivarEspera) THEN
       #Apil_ET05 := TRUE;   // SR flip-flop
   END_IF;
   IF #Apil_ET06 THEN #Apil_ET05 := FALSE; END_IF;
END_REGION

REGION Network 30: --- TIM Espera ET05
   RUNG wire#powerrail
      Contact( #Apil_ET04 )
      Contact( #CentradoresAbiertos )
      Contact( #Carga_PosicionIntermedia )
      I_Contact( #OrdenMover )
      I_Contact( #Fin_OrdenMover )
      I_Contact( #MemoPosicionOK )
      { S7_Templates := "time_type := Time" } #TIM_EsperaET05.TON(pt := T#100ms, et =>)
   END_RUNG
   // the same network as SCL:
   #TIM_EsperaET05(IN := #Apil_ET04 AND #CentradoresAbiertos AND #Carga_PosicionIntermedia AND NOT #OrdenMover AND NOT #Fin_OrdenMover AND NOT #MemoPosicionOK,   // TON
                   PT := T#100ms);
END_REGION

REGION Network 31: Apil_ET04
   // Cerradas las Garras
   RUNG wire#powerrail
      Contact( #Apil_ET03 )
      wire#w1
      Contact( #GarrasCerradas )
      I_Contact( #OrdenMover )
      I_Contact( #Fin_OrdenMover )
      I_Contact( #MemoPosicionOK )
      wire#w2
      S_SR(operand := #Apil_ET04, r1 := #Apil_ET05)
   END_RUNG
   RUNG wire#w1
      I_Contact( #pHsMx_PresCarga )
      I_Contact( #OrdenMover )
      I_Contact( #Fin_OrdenMover )
      I_Contact( #MemoPosicionOK )
   END_RUNG wire#w2
   // the same network as SCL:
   IF #Apil_ET03 AND ((#GarrasCerradas AND NOT #OrdenMover AND NOT #Fin_OrdenMover AND NOT #MemoPosicionOK) OR (NOT #pHsMx_PresCarga AND NOT #OrdenMover AND NOT #Fin_OrdenMover AND NOT #MemoPosicionOK)) THEN
       #Apil_ET04 := TRUE;   // SR flip-flop
   END_IF;
   IF #Apil_ET05 THEN #Apil_ET04 := FALSE; END_IF;
END_REGION

REGION Network 32: Apil_ET03
   // Posicionado en la PosInicial
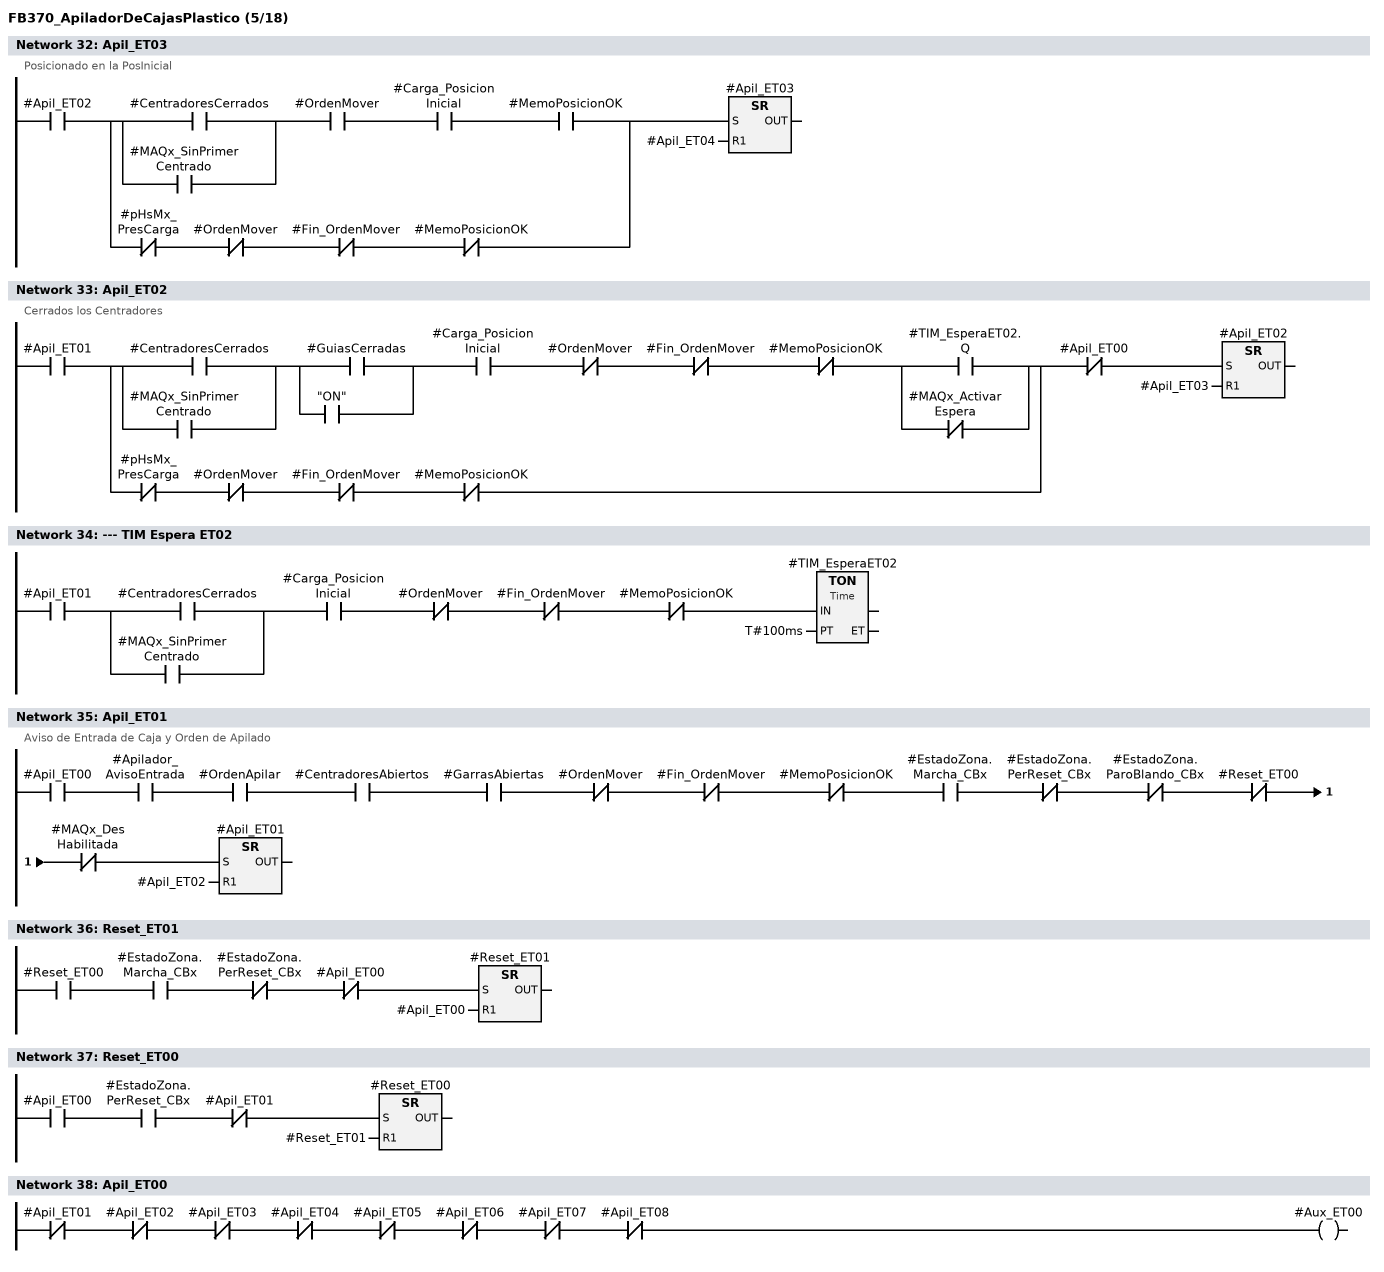
   RUNG wire#powerrail
      Contact( #Apil_ET02 )
      wire#w1
      Contact( #CentradoresCerrados )
      wire#w2
      Contact( #OrdenMover )
      Contact( #Carga_PosicionInicial )
      Contact( #MemoPosicionOK )
      wire#w3
      S_SR(operand := #Apil_ET03, r1 := #Apil_ET04)
   END_RUNG
   RUNG wire#w1
      Contact( #MAQx_SinPrimerCentrado )
   END_RUNG wire#w2
   RUNG wire#w1
      I_Contact( #pHsMx_PresCarga )
      I_Contact( #OrdenMover )
      I_Contact( #Fin_OrdenMover )
      I_Contact( #MemoPosicionOK )
   END_RUNG wire#w3
   // the same network as SCL:
   IF #Apil_ET02 AND (((#CentradoresCerrados OR #MAQx_SinPrimerCentrado) AND #OrdenMover AND #Carga_PosicionInicial AND #MemoPosicionOK) OR (NOT #pHsMx_PresCarga AND NOT #OrdenMover AND NOT #Fin_OrdenMover AND NOT #MemoPosicionOK)) THEN
       #Apil_ET03 := TRUE;   // SR flip-flop
   END_IF;
   IF #Apil_ET04 THEN #Apil_ET03 := FALSE; END_IF;
END_REGION

REGION Network 33: Apil_ET02
   // Cerrados los Centradores
   RUNG wire#powerrail
      Contact( #Apil_ET01 )
      wire#w1
      Contact( #CentradoresCerrados )
      wire#w2
      Contact( #GuiasCerradas )
      wire#w3
      Contact( #Carga_PosicionInicial )
      I_Contact( #OrdenMover )
      I_Contact( #Fin_OrdenMover )
      I_Contact( #MemoPosicionOK )
      wire#w4
      Contact( #TIM_EsperaET02.Q )
      wire#w5
      I_Contact( #Apil_ET00 )
      S_SR(operand := #Apil_ET02, r1 := #Apil_ET03)
   END_RUNG
   RUNG wire#w1
      Contact( #MAQx_SinPrimerCentrado )
   END_RUNG wire#w2
   RUNG wire#w2
      Contact( "ON" )
   END_RUNG wire#w3
   RUNG wire#w4
      I_Contact( #MAQx_ActivarEspera )
   END_RUNG wire#w5
   RUNG wire#w1
      I_Contact( #pHsMx_PresCarga )
      I_Contact( #OrdenMover )
      I_Contact( #Fin_OrdenMover )
      I_Contact( #MemoPosicionOK )
   END_RUNG wire#w5
   // the same network as SCL:
   IF #Apil_ET01 AND (((#CentradoresCerrados OR #MAQx_SinPrimerCentrado) AND (#GuiasCerradas OR "ON") AND #Carga_PosicionInicial AND NOT #OrdenMover AND NOT #Fin_OrdenMover AND NOT #MemoPosicionOK AND (#TIM_EsperaET02.Q OR NOT #MAQx_ActivarEspera)) OR (NOT #pHsMx_PresCarga AND NOT #OrdenMover AND NOT #Fin_OrdenMover AND NOT #MemoPosicionOK)) AND NOT #Apil_ET00 THEN
       #Apil_ET02 := TRUE;   // SR flip-flop
   END_IF;
   IF #Apil_ET03 THEN #Apil_ET02 := FALSE; END_IF;
END_REGION

REGION Network 34: --- TIM Espera ET02
   RUNG wire#powerrail
      Contact( #Apil_ET01 )
      wire#w1
      Contact( #CentradoresCerrados )
      wire#w2
      Contact( #Carga_PosicionInicial )
      I_Contact( #OrdenMover )
      I_Contact( #Fin_OrdenMover )
      I_Contact( #MemoPosicionOK )
      { S7_Templates := "time_type := Time" } #TIM_EsperaET02.TON(pt := T#100ms, et =>)
   END_RUNG
   RUNG wire#w1
      Contact( #MAQx_SinPrimerCentrado )
   END_RUNG wire#w2
   // the same network as SCL:
   #TIM_EsperaET02(IN := #Apil_ET01 AND (#CentradoresCerrados OR #MAQx_SinPrimerCentrado) AND #Carga_PosicionInicial AND NOT #OrdenMover AND NOT #Fin_OrdenMover AND NOT #MemoPosicionOK,   // TON
                   PT := T#100ms);
END_REGION

REGION Network 35: Apil_ET01
   // Aviso de Entrada de Caja y Orden de Apilado
   RUNG wire#powerrail
      Contact( #Apil_ET00 )
      Contact( #Apilador_AvisoEntrada )
      Contact( #OrdenApilar )
      Contact( #CentradoresAbiertos )
      Contact( #GarrasAbiertas )
      I_Contact( #OrdenMover )
      I_Contact( #Fin_OrdenMover )
      I_Contact( #MemoPosicionOK )
      Contact( #EstadoZona.Marcha_CBx )
      I_Contact( #EstadoZona.PerReset_CBx )
      I_Contact( #EstadoZona.ParoBlando_CBx )
      I_Contact( #Reset_ET00 )
      I_Contact( #MAQx_DesHabilitada )
      S_SR(operand := #Apil_ET01, r1 := #Apil_ET02)
   END_RUNG
   // the same network as SCL:
   IF #Apil_ET00 AND #Apilador_AvisoEntrada AND #OrdenApilar AND #CentradoresAbiertos AND #GarrasAbiertas AND NOT #OrdenMover AND NOT #Fin_OrdenMover AND NOT #MemoPosicionOK AND #EstadoZona.Marcha_CBx AND NOT #EstadoZona.PerReset_CBx AND NOT #EstadoZona.ParoBlando_CBx AND NOT #Reset_ET00 AND NOT #MAQx_DesHabilitada THEN
       #Apil_ET01 := TRUE;   // SR flip-flop
   END_IF;
   IF #Apil_ET02 THEN #Apil_ET01 := FALSE; END_IF;
END_REGION

REGION Network 36: Reset_ET01
   RUNG wire#powerrail
      Contact( #Reset_ET00 )
      Contact( #EstadoZona.Marcha_CBx )
      I_Contact( #EstadoZona.PerReset_CBx )
      I_Contact( #Apil_ET00 )
      S_SR(operand := #Reset_ET01, r1 := #Apil_ET00)
   END_RUNG
   // the same network as SCL:
   IF #Reset_ET00 AND #EstadoZona.Marcha_CBx AND NOT #EstadoZona.PerReset_CBx AND NOT #Apil_ET00 THEN
       #Reset_ET01 := TRUE;   // SR flip-flop
   END_IF;
   IF #Apil_ET00 THEN #Reset_ET01 := FALSE; END_IF;
END_REGION

REGION Network 37: Reset_ET00
   RUNG wire#powerrail
      Contact( #Apil_ET00 )
      Contact( #EstadoZona.PerReset_CBx )
      I_Contact( #Apil_ET01 )
      S_SR(operand := #Reset_ET00, r1 := #Reset_ET01)
   END_RUNG
   // the same network as SCL:
   IF #Apil_ET00 AND #EstadoZona.PerReset_CBx AND NOT #Apil_ET01 THEN
       #Reset_ET00 := TRUE;   // SR flip-flop
   END_IF;
   IF #Reset_ET01 THEN #Reset_ET00 := FALSE; END_IF;
END_REGION

REGION Network 38: Apil_ET00
   RUNG wire#powerrail
      I_Contact( #Apil_ET01 )
      I_Contact( #Apil_ET02 )
      I_Contact( #Apil_ET03 )
      I_Contact( #Apil_ET04 )
      I_Contact( #Apil_ET05 )
      I_Contact( #Apil_ET06 )
      I_Contact( #Apil_ET07 )
      I_Contact( #Apil_ET08 )
      Coil( #Aux_ET00 )
   END_RUNG
   // the same network as SCL:
   #Aux_ET00 := NOT #Apil_ET01 AND NOT #Apil_ET02 AND NOT #Apil_ET03 AND NOT #Apil_ET04 AND NOT #Apil_ET05 AND NOT #Apil_ET06 AND NOT #Apil_ET07 AND NOT #Apil_ET08;
END_REGION

REGION Network 39: ---
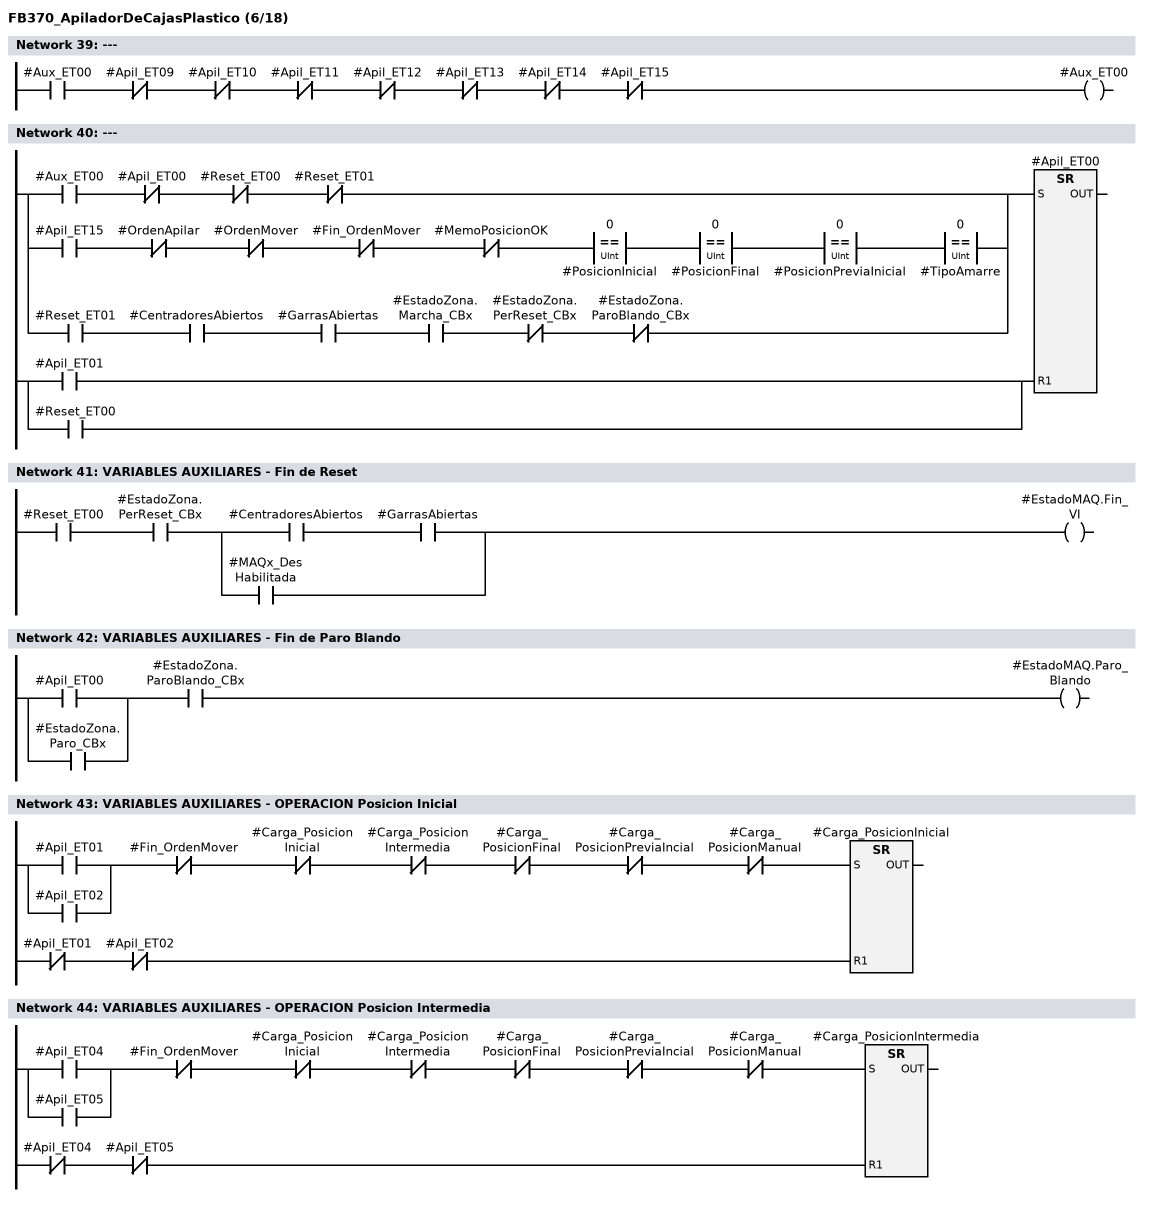
   RUNG wire#powerrail
      Contact( #Aux_ET00 )
      I_Contact( #Apil_ET09 )
      I_Contact( #Apil_ET10 )
      I_Contact( #Apil_ET11 )
      I_Contact( #Apil_ET12 )
      I_Contact( #Apil_ET13 )
      I_Contact( #Apil_ET14 )
      I_Contact( #Apil_ET15 )
      Coil( #Aux_ET00 )
   END_RUNG
   // the same network as SCL:
   #Aux_ET00 := #Aux_ET00 AND NOT #Apil_ET09 AND NOT #Apil_ET10 AND NOT #Apil_ET11 AND NOT #Apil_ET12 AND NOT #Apil_ET13 AND NOT #Apil_ET14 AND NOT #Apil_ET15;
END_REGION

REGION Network 40: ---
   RUNG wire#powerrail
      Contact( #Aux_ET00 )
      I_Contact( #Apil_ET00 )
      I_Contact( #Reset_ET00 )
      I_Contact( #Reset_ET01 )
      wire#w1
      S_SR(operand := #Apil_ET00, r1 := wire#w2)
   END_RUNG
   RUNG wire#powerrail
      Contact( #Apil_ET15 )
      I_Contact( #OrdenApilar )
      I_Contact( #OrdenMover )
      I_Contact( #Fin_OrdenMover )
      I_Contact( #MemoPosicionOK )
      { S7_Templates := "SrcType := UInt" } EQ_Contact(in1 := 0, in2 := #PosicionInicial)
      { S7_Templates := "SrcType := UInt" } EQ_Contact(in1 := 0, in2 := #PosicionFinal)
      { S7_Templates := "SrcType := UInt" } EQ_Contact(in1 := 0, in2 := #PosicionPreviaInicial)
      { S7_Templates := "SrcType := UInt" } EQ_Contact(in1 := 0, in2 := #TipoAmarre)
   END_RUNG wire#w1
   RUNG wire#powerrail
      Contact( #Reset_ET01 )
      Contact( #CentradoresAbiertos )
      Contact( #GarrasAbiertas )
      Contact( #EstadoZona.Marcha_CBx )
      I_Contact( #EstadoZona.PerReset_CBx )
      I_Contact( #EstadoZona.ParoBlando_CBx )
   END_RUNG wire#w1
   RUNG wire#powerrail
      Contact( #Apil_ET01 )
   END_RUNG wire#w2
   RUNG wire#powerrail
      Contact( #Reset_ET00 )
   END_RUNG wire#w2
   // the same network as SCL:
   IF (#Aux_ET00 AND NOT #Apil_ET00 AND NOT #Reset_ET00 AND NOT #Reset_ET01) OR (#Apil_ET15 AND NOT #OrdenApilar AND NOT #OrdenMover AND NOT #Fin_OrdenMover AND NOT #MemoPosicionOK AND (0 = #PosicionInicial) AND (0 = #PosicionFinal) AND (0 = #PosicionPreviaInicial) AND (0 = #TipoAmarre)) OR (#Reset_ET01 AND #CentradoresAbiertos AND #GarrasAbiertas AND #EstadoZona.Marcha_CBx AND NOT #EstadoZona.PerReset_CBx AND NOT #EstadoZona.ParoBlando_CBx) THEN
       #Apil_ET00 := TRUE;   // SR flip-flop
   END_IF;
   IF #Apil_ET01 OR #Reset_ET00 THEN #Apil_ET00 := FALSE; END_IF;
END_REGION

REGION Network 41: VARIABLES AUXILIARES - Fin de Reset
   RUNG wire#powerrail
      Contact( #Reset_ET00 )
      Contact( #EstadoZona.PerReset_CBx )
      wire#w1
      Contact( #CentradoresAbiertos )
      Contact( #GarrasAbiertas )
      wire#w2
      Coil( #EstadoMAQ.Fin_VI )
   END_RUNG
   RUNG wire#w1
      Contact( #MAQx_DesHabilitada )
   END_RUNG wire#w2
   // the same network as SCL:
   #EstadoMAQ.Fin_VI := #Reset_ET00 AND #EstadoZona.PerReset_CBx AND ((#CentradoresAbiertos AND #GarrasAbiertas) OR #MAQx_DesHabilitada);
END_REGION

REGION Network 42: VARIABLES AUXILIARES - Fin de Paro Blando
   RUNG wire#powerrail
      Contact( #Apil_ET00 )
      wire#w1
      Contact( #EstadoZona.ParoBlando_CBx )
      Coil( #EstadoMAQ.Paro_Blando )
   END_RUNG
   RUNG wire#powerrail
      Contact( #EstadoZona.Paro_CBx )
   END_RUNG wire#w1
   // the same network as SCL:
   #EstadoMAQ.Paro_Blando := (#Apil_ET00 OR #EstadoZona.Paro_CBx) AND #EstadoZona.ParoBlando_CBx;
END_REGION

REGION Network 43: VARIABLES AUXILIARES - OPERACION Posicion Inicial
   RUNG wire#powerrail
      Contact( #Apil_ET01 )
      wire#w1
      I_Contact( #Fin_OrdenMover )
      I_Contact( #Carga_PosicionInicial )
      I_Contact( #Carga_PosicionIntermedia )
      I_Contact( #Carga_PosicionFinal )
      I_Contact( #Carga_PosicionPreviaIncial )
      I_Contact( #Carga_PosicionManual )
      S_SR(operand := #Carga_PosicionInicial, r1 := wire#w2)
   END_RUNG
   RUNG wire#powerrail
      Contact( #Apil_ET02 )
   END_RUNG wire#w1
   RUNG wire#powerrail
      I_Contact( #Apil_ET01 )
      I_Contact( #Apil_ET02 )
   END_RUNG wire#w2
   // the same network as SCL:
   IF (#Apil_ET01 OR #Apil_ET02) AND NOT #Fin_OrdenMover AND NOT #Carga_PosicionInicial AND NOT #Carga_PosicionIntermedia AND NOT #Carga_PosicionFinal AND NOT #Carga_PosicionPreviaIncial AND NOT #Carga_PosicionManual THEN
       #Carga_PosicionInicial := TRUE;   // SR flip-flop
   END_IF;
   IF NOT #Apil_ET01 AND NOT #Apil_ET02 THEN #Carga_PosicionInicial := FALSE; END_IF;
END_REGION

REGION Network 44: VARIABLES AUXILIARES - OPERACION Posicion Intermedia
   RUNG wire#powerrail
      Contact( #Apil_ET04 )
      wire#w1
      I_Contact( #Fin_OrdenMover )
      I_Contact( #Carga_PosicionInicial )
      I_Contact( #Carga_PosicionIntermedia )
      I_Contact( #Carga_PosicionFinal )
      I_Contact( #Carga_PosicionPreviaIncial )
      I_Contact( #Carga_PosicionManual )
      S_SR(operand := #Carga_PosicionIntermedia, r1 := wire#w2)
   END_RUNG
   RUNG wire#powerrail
      Contact( #Apil_ET05 )
   END_RUNG wire#w1
   RUNG wire#powerrail
      I_Contact( #Apil_ET04 )
      I_Contact( #Apil_ET05 )
   END_RUNG wire#w2
   // the same network as SCL:
   IF (#Apil_ET04 OR #Apil_ET05) AND NOT #Fin_OrdenMover AND NOT #Carga_PosicionInicial AND NOT #Carga_PosicionIntermedia AND NOT #Carga_PosicionFinal AND NOT #Carga_PosicionPreviaIncial AND NOT #Carga_PosicionManual THEN
       #Carga_PosicionIntermedia := TRUE;   // SR flip-flop
   END_IF;
   IF NOT #Apil_ET04 AND NOT #Apil_ET05 THEN #Carga_PosicionIntermedia := FALSE; END_IF;
END_REGION

REGION Network 45: VARIABLES AUXILIARES - OPERACION Posicion Final
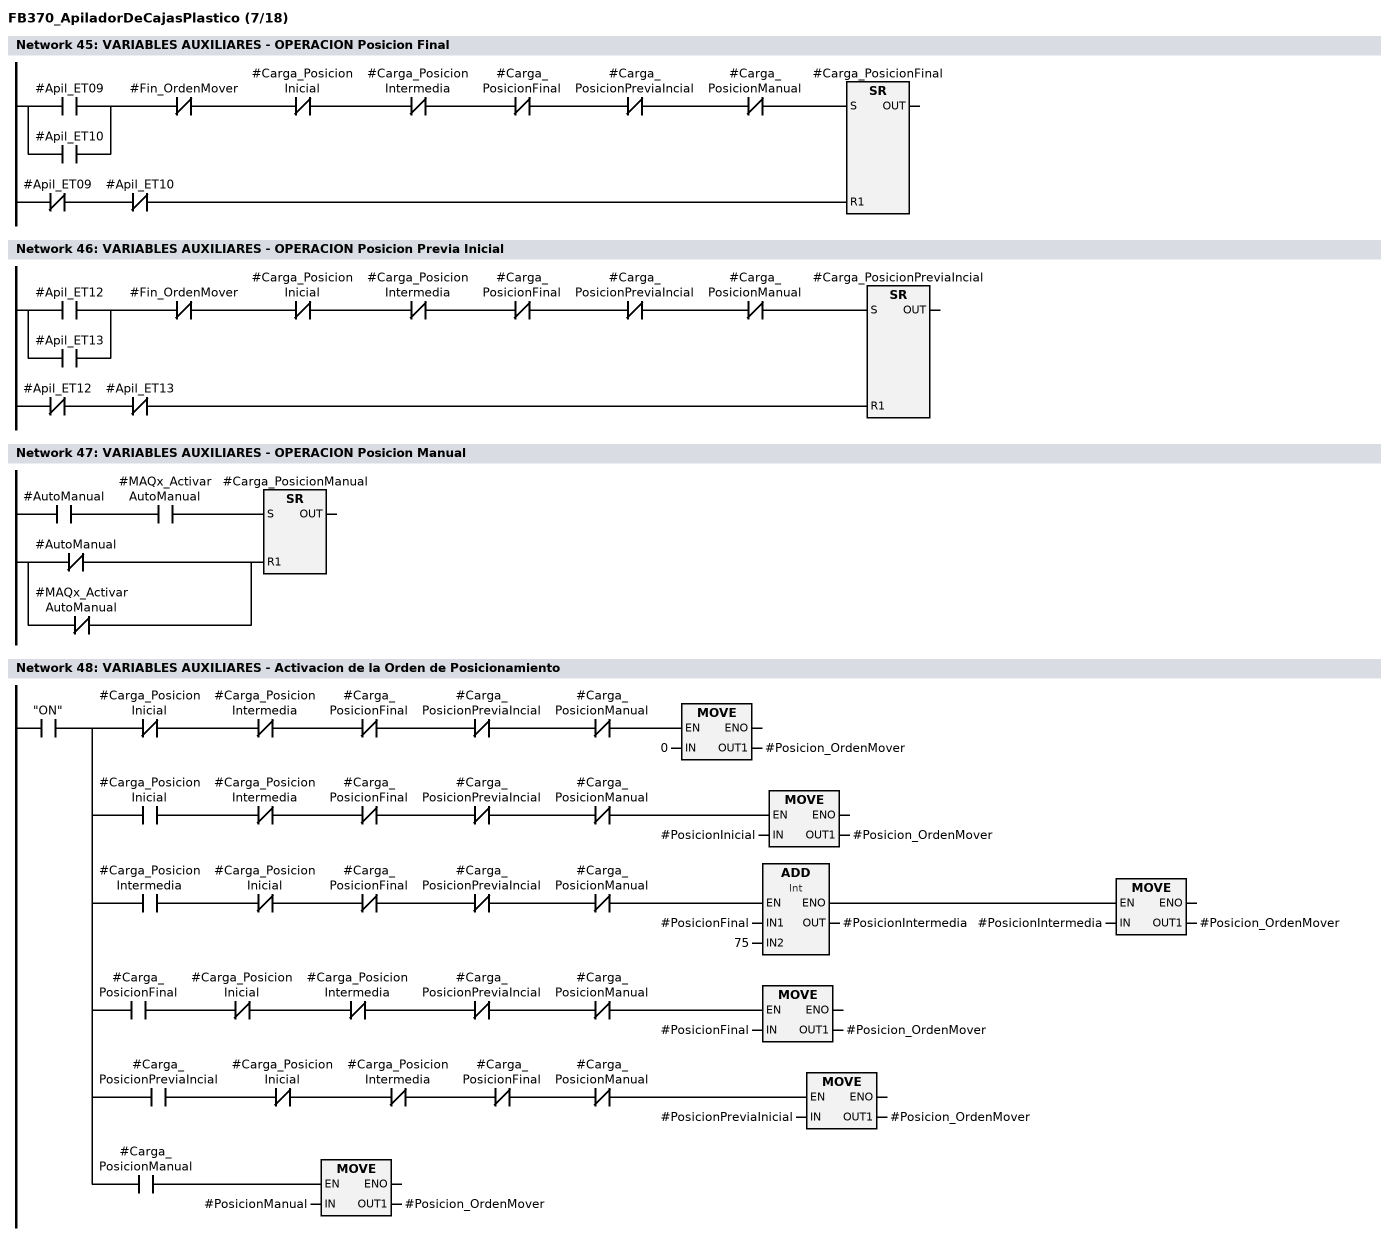
   RUNG wire#powerrail
      Contact( #Apil_ET09 )
      wire#w1
      I_Contact( #Fin_OrdenMover )
      I_Contact( #Carga_PosicionInicial )
      I_Contact( #Carga_PosicionIntermedia )
      I_Contact( #Carga_PosicionFinal )
      I_Contact( #Carga_PosicionPreviaIncial )
      I_Contact( #Carga_PosicionManual )
      S_SR(operand := #Carga_PosicionFinal, r1 := wire#w2)
   END_RUNG
   RUNG wire#powerrail
      Contact( #Apil_ET10 )
   END_RUNG wire#w1
   RUNG wire#powerrail
      I_Contact( #Apil_ET09 )
      I_Contact( #Apil_ET10 )
   END_RUNG wire#w2
   // the same network as SCL:
   IF (#Apil_ET09 OR #Apil_ET10) AND NOT #Fin_OrdenMover AND NOT #Carga_PosicionInicial AND NOT #Carga_PosicionIntermedia AND NOT #Carga_PosicionFinal AND NOT #Carga_PosicionPreviaIncial AND NOT #Carga_PosicionManual THEN
       #Carga_PosicionFinal := TRUE;   // SR flip-flop
   END_IF;
   IF NOT #Apil_ET09 AND NOT #Apil_ET10 THEN #Carga_PosicionFinal := FALSE; END_IF;
END_REGION

REGION Network 46: VARIABLES AUXILIARES - OPERACION Posicion Previa Inicial
   RUNG wire#powerrail
      Contact( #Apil_ET12 )
      wire#w1
      I_Contact( #Fin_OrdenMover )
      I_Contact( #Carga_PosicionInicial )
      I_Contact( #Carga_PosicionIntermedia )
      I_Contact( #Carga_PosicionFinal )
      I_Contact( #Carga_PosicionPreviaIncial )
      I_Contact( #Carga_PosicionManual )
      S_SR(operand := #Carga_PosicionPreviaIncial, r1 := wire#w2)
   END_RUNG
   RUNG wire#powerrail
      Contact( #Apil_ET13 )
   END_RUNG wire#w1
   RUNG wire#powerrail
      I_Contact( #Apil_ET12 )
      I_Contact( #Apil_ET13 )
   END_RUNG wire#w2
   // the same network as SCL:
   IF (#Apil_ET12 OR #Apil_ET13) AND NOT #Fin_OrdenMover AND NOT #Carga_PosicionInicial AND NOT #Carga_PosicionIntermedia AND NOT #Carga_PosicionFinal AND NOT #Carga_PosicionPreviaIncial AND NOT #Carga_PosicionManual THEN
       #Carga_PosicionPreviaIncial := TRUE;   // SR flip-flop
   END_IF;
   IF NOT #Apil_ET12 AND NOT #Apil_ET13 THEN #Carga_PosicionPreviaIncial := FALSE; END_IF;
END_REGION

REGION Network 47: VARIABLES AUXILIARES - OPERACION Posicion Manual
   RUNG wire#powerrail
      Contact( #AutoManual )
      Contact( #MAQx_ActivarAutoManual )
      S_SR(operand := #Carga_PosicionManual, r1 := wire#w1)
   END_RUNG
   RUNG wire#powerrail
      I_Contact( #AutoManual )
   END_RUNG wire#w1
   RUNG wire#powerrail
      I_Contact( #MAQx_ActivarAutoManual )
   END_RUNG wire#w1
   // the same network as SCL:
   IF #AutoManual AND #MAQx_ActivarAutoManual THEN
       #Carga_PosicionManual := TRUE;   // SR flip-flop
   END_IF;
   IF NOT #AutoManual OR NOT #MAQx_ActivarAutoManual THEN #Carga_PosicionManual := FALSE; END_IF;
END_REGION

REGION Network 48: VARIABLES AUXILIARES - Activacion de la Orden de Posicionamiento
   RUNG wire#powerrail
      Contact( "ON" )
      wire#w1
      I_Contact( #Carga_PosicionInicial )
      I_Contact( #Carga_PosicionIntermedia )
      I_Contact( #Carga_PosicionFinal )
      I_Contact( #Carga_PosicionPreviaIncial )
      I_Contact( #Carga_PosicionManual )
      { S7_GenerateENO := "TRUE" } Move(in := 0, out1 => #Posicion_OrdenMover)
   END_RUNG
   RUNG wire#w1
      Contact( #Carga_PosicionInicial )
      I_Contact( #Carga_PosicionIntermedia )
      I_Contact( #Carga_PosicionFinal )
      I_Contact( #Carga_PosicionPreviaIncial )
      I_Contact( #Carga_PosicionManual )
      { S7_GenerateENO := "TRUE" } Move(in := #PosicionInicial, out1 => #Posicion_OrdenMover)
   END_RUNG
   RUNG wire#w1
      Contact( #Carga_PosicionIntermedia )
      I_Contact( #Carga_PosicionInicial )
      I_Contact( #Carga_PosicionFinal )
      I_Contact( #Carga_PosicionPreviaIncial )
      I_Contact( #Carga_PosicionManual )
      { S7_Templates := "SrcType := Int"; S7_GenerateENO := "TRUE" } Add(in1 := #PosicionFinal, in2 := 75, out => #PosicionIntermedia)
      { S7_GenerateENO := "TRUE" } Move(in := #PosicionIntermedia, out1 => #Posicion_OrdenMover)
   END_RUNG
   RUNG wire#w1
      Contact( #Carga_PosicionFinal )
      I_Contact( #Carga_PosicionInicial )
      I_Contact( #Carga_PosicionIntermedia )
      I_Contact( #Carga_PosicionPreviaIncial )
      I_Contact( #Carga_PosicionManual )
      { S7_GenerateENO := "TRUE" } Move(in := #PosicionFinal, out1 => #Posicion_OrdenMover)
   END_RUNG
   RUNG wire#w1
      Contact( #Carga_PosicionPreviaIncial )
      I_Contact( #Carga_PosicionInicial )
      I_Contact( #Carga_PosicionIntermedia )
      I_Contact( #Carga_PosicionFinal )
      I_Contact( #Carga_PosicionManual )
      { S7_GenerateENO := "TRUE" } Move(in := #PosicionPreviaInicial, out1 => #Posicion_OrdenMover)
   END_RUNG
   RUNG wire#w1
      Contact( #Carga_PosicionManual )
      { S7_GenerateENO := "TRUE" } Move(in := #PosicionManual, out1 => #Posicion_OrdenMover)
   END_RUNG
   // the same network as SCL:
   // ENO of a box is taken as its EN; it also drops when the box reports an error
   IF "ON" AND NOT #Carga_PosicionInicial AND NOT #Carga_PosicionIntermedia AND NOT #Carga_PosicionFinal AND NOT #Carga_PosicionPreviaIncial AND NOT #Carga_PosicionManual THEN
       #Posicion_OrdenMover := 0;
   END_IF;
   IF "ON" AND #Carga_PosicionInicial AND NOT #Carga_PosicionIntermedia AND NOT #Carga_PosicionFinal AND NOT #Carga_PosicionPreviaIncial AND NOT #Carga_PosicionManual THEN
       #Posicion_OrdenMover := #PosicionInicial;
   END_IF;
   IF "ON" AND #Carga_PosicionIntermedia AND NOT #Carga_PosicionInicial AND NOT #Carga_PosicionFinal AND NOT #Carga_PosicionPreviaIncial AND NOT #Carga_PosicionManual THEN
       #PosicionIntermedia := #PosicionFinal + 75;
       #Posicion_OrdenMover := #PosicionIntermedia;
   END_IF;
   IF "ON" AND #Carga_PosicionFinal AND NOT #Carga_PosicionInicial AND NOT #Carga_PosicionIntermedia AND NOT #Carga_PosicionPreviaIncial AND NOT #Carga_PosicionManual THEN
       #Posicion_OrdenMover := #PosicionFinal;
   END_IF;
   IF "ON" AND #Carga_PosicionPreviaIncial AND NOT #Carga_PosicionInicial AND NOT #Carga_PosicionIntermedia AND NOT #Carga_PosicionFinal AND NOT #Carga_PosicionManual THEN
       #Posicion_OrdenMover := #PosicionPreviaInicial;
   END_IF;
   IF "ON" AND #Carga_PosicionManual THEN #Posicion_OrdenMover := #PosicionManual; END_IF;
END_REGION

REGION Network 49: ---
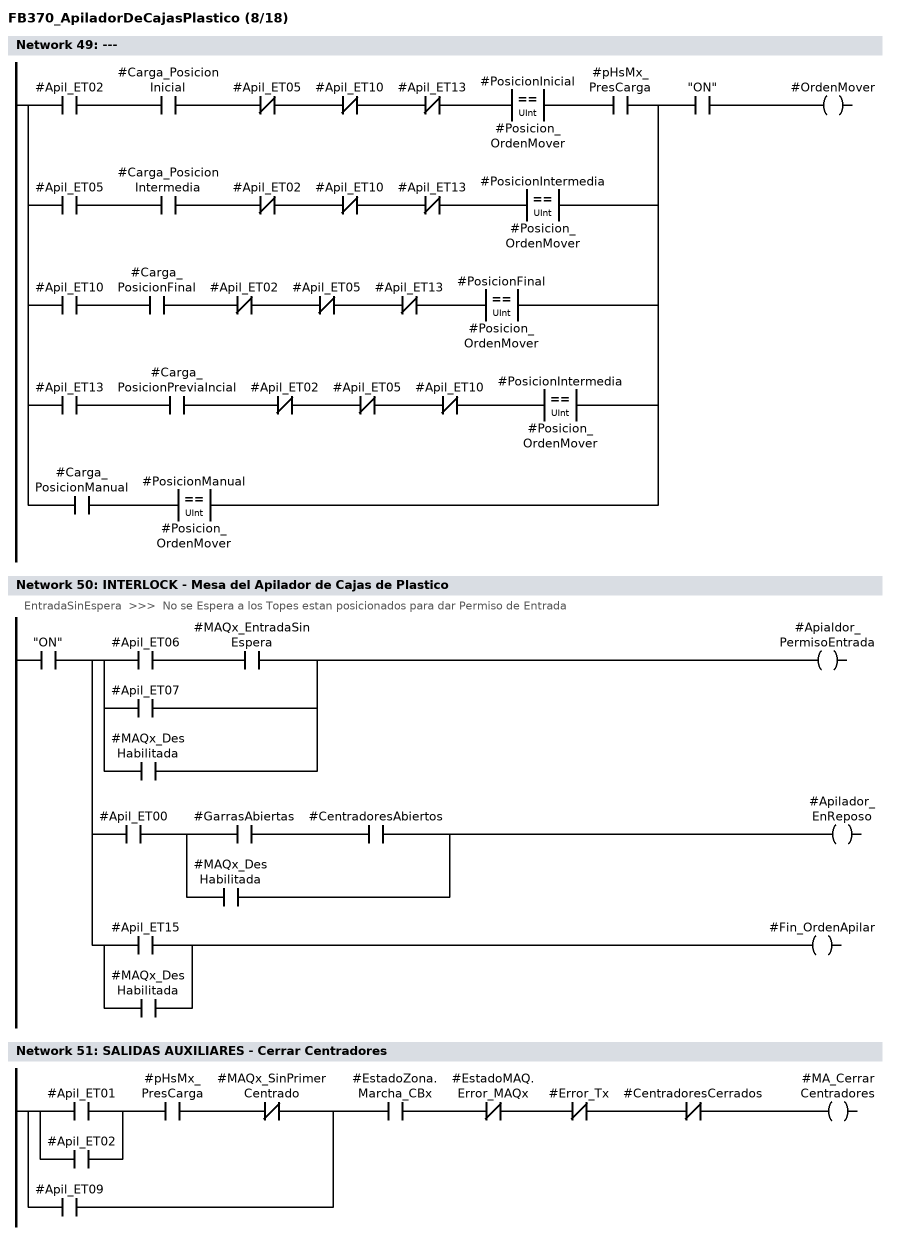
   RUNG wire#powerrail
      Contact( #Apil_ET02 )
      Contact( #Carga_PosicionInicial )
      I_Contact( #Apil_ET05 )
      I_Contact( #Apil_ET10 )
      I_Contact( #Apil_ET13 )
      { S7_Templates := "SrcType := UInt" } EQ_Contact(in1 := #PosicionInicial, in2 := #Posicion_OrdenMover)
      Contact( #pHsMx_PresCarga )
      wire#w1
      Contact( "ON" )
      Coil( #OrdenMover )
   END_RUNG
   RUNG wire#powerrail
      Contact( #Apil_ET05 )
      Contact( #Carga_PosicionIntermedia )
      I_Contact( #Apil_ET02 )
      I_Contact( #Apil_ET10 )
      I_Contact( #Apil_ET13 )
      { S7_Templates := "SrcType := UInt" } EQ_Contact(in1 := #PosicionIntermedia, in2 := #Posicion_OrdenMover)
   END_RUNG wire#w1
   RUNG wire#powerrail
      Contact( #Apil_ET10 )
      Contact( #Carga_PosicionFinal )
      I_Contact( #Apil_ET02 )
      I_Contact( #Apil_ET05 )
      I_Contact( #Apil_ET13 )
      { S7_Templates := "SrcType := UInt" } EQ_Contact(in1 := #PosicionFinal, in2 := #Posicion_OrdenMover)
   END_RUNG wire#w1
   RUNG wire#powerrail
      Contact( #Apil_ET13 )
      Contact( #Carga_PosicionPreviaIncial )
      I_Contact( #Apil_ET02 )
      I_Contact( #Apil_ET05 )
      I_Contact( #Apil_ET10 )
      { S7_Templates := "SrcType := UInt" } EQ_Contact(in1 := #PosicionIntermedia, in2 := #Posicion_OrdenMover)
   END_RUNG wire#w1
   RUNG wire#powerrail
      Contact( #Carga_PosicionManual )
      { S7_Templates := "SrcType := UInt" } EQ_Contact(in1 := #PosicionManual, in2 := #Posicion_OrdenMover)
   END_RUNG wire#w1
   // the same network as SCL:
   #OrdenMover := ((#Apil_ET02 AND #Carga_PosicionInicial AND NOT #Apil_ET05 AND NOT #Apil_ET10 AND NOT #Apil_ET13 AND (#PosicionInicial = #Posicion_OrdenMover) AND #pHsMx_PresCarga) OR (#Apil_ET05 AND #Carga_PosicionIntermedia AND NOT #Apil_ET02 AND NOT #Apil_ET10 AND NOT #Apil_ET13 AND (#PosicionIntermedia = #Posicion_OrdenMover)) OR (#Apil_ET10 AND #Carga_PosicionFinal AND NOT #Apil_ET02 AND NOT #Apil_ET05 AND NOT #Apil_ET13 AND (#PosicionFinal = #Posicion_OrdenMover)) OR (#Apil_ET13 AND #Carga_PosicionPreviaIncial AND NOT #Apil_ET02 AND NOT #Apil_ET05 AND NOT #Apil_ET10 AND (#PosicionIntermedia = #Posicion_OrdenMover)) OR (#Carga_PosicionManual AND (#PosicionManual = #Posicion_OrdenMover))) AND "ON";
END_REGION

REGION Network 50: INTERLOCK - Mesa del Apilador de Cajas de Plastico
   // EntradaSinEspera  >>>  No se Espera a los Topes estan posicionados para dar Permiso de Entrada
   RUNG wire#powerrail
      Contact( "ON" )
      wire#w1
      Contact( #Apil_ET06 )
      Contact( #MAQx_EntradaSinEspera )
      wire#w2
      Coil( #Apialdor_PermisoEntrada )
   END_RUNG
   RUNG wire#w1
      Contact( #Apil_ET07 )
   END_RUNG wire#w2
   RUNG wire#w1
      Contact( #MAQx_DesHabilitada )
   END_RUNG wire#w2
   RUNG wire#w1
      Contact( #Apil_ET00 )
      wire#w3
      Contact( #GarrasAbiertas )
      Contact( #CentradoresAbiertos )
      wire#w4
      Coil( #Apilador_EnReposo )
   END_RUNG
   RUNG wire#w3
      Contact( #MAQx_DesHabilitada )
   END_RUNG wire#w4
   RUNG wire#w1
      Contact( #Apil_ET15 )
      wire#w5
      Coil( #Fin_OrdenApilar )
   END_RUNG
   RUNG wire#w1
      Contact( #MAQx_DesHabilitada )
   END_RUNG wire#w5
   // the same network as SCL:
   #Apialdor_PermisoEntrada := "ON" AND ((#Apil_ET06 AND #MAQx_EntradaSinEspera) OR #Apil_ET07 OR #MAQx_DesHabilitada);
   #Apilador_EnReposo := "ON" AND #Apil_ET00 AND ((#GarrasAbiertas AND #CentradoresAbiertos) OR #MAQx_DesHabilitada);
   #Fin_OrdenApilar := "ON" AND (#Apil_ET15 OR #MAQx_DesHabilitada);
END_REGION

REGION Network 51: SALIDAS AUXILIARES - Cerrar Centradores
   RUNG wire#powerrail
      Contact( #Apil_ET01 )
      wire#w1
      Contact( #pHsMx_PresCarga )
      I_Contact( #MAQx_SinPrimerCentrado )
      wire#w2
      Contact( #EstadoZona.Marcha_CBx )
      I_Contact( #EstadoMAQ.Error_MAQx )
      I_Contact( #Error_Tx )
      I_Contact( #CentradoresCerrados )
      Coil( #MA_CerrarCentradores )
   END_RUNG
   RUNG wire#powerrail
      Contact( #Apil_ET02 )
   END_RUNG wire#w1
   RUNG wire#powerrail
      Contact( #Apil_ET09 )
   END_RUNG wire#w2
   // the same network as SCL:
   #MA_CerrarCentradores := (((#Apil_ET01 OR #Apil_ET02) AND #pHsMx_PresCarga AND NOT #MAQx_SinPrimerCentrado) OR #Apil_ET09) AND #EstadoZona.Marcha_CBx AND NOT #EstadoMAQ.Error_MAQx AND NOT #Error_Tx AND NOT #CentradoresCerrados;
END_REGION

REGION Network 52: SALIDAS AUXILIARES - Abrir Centradores
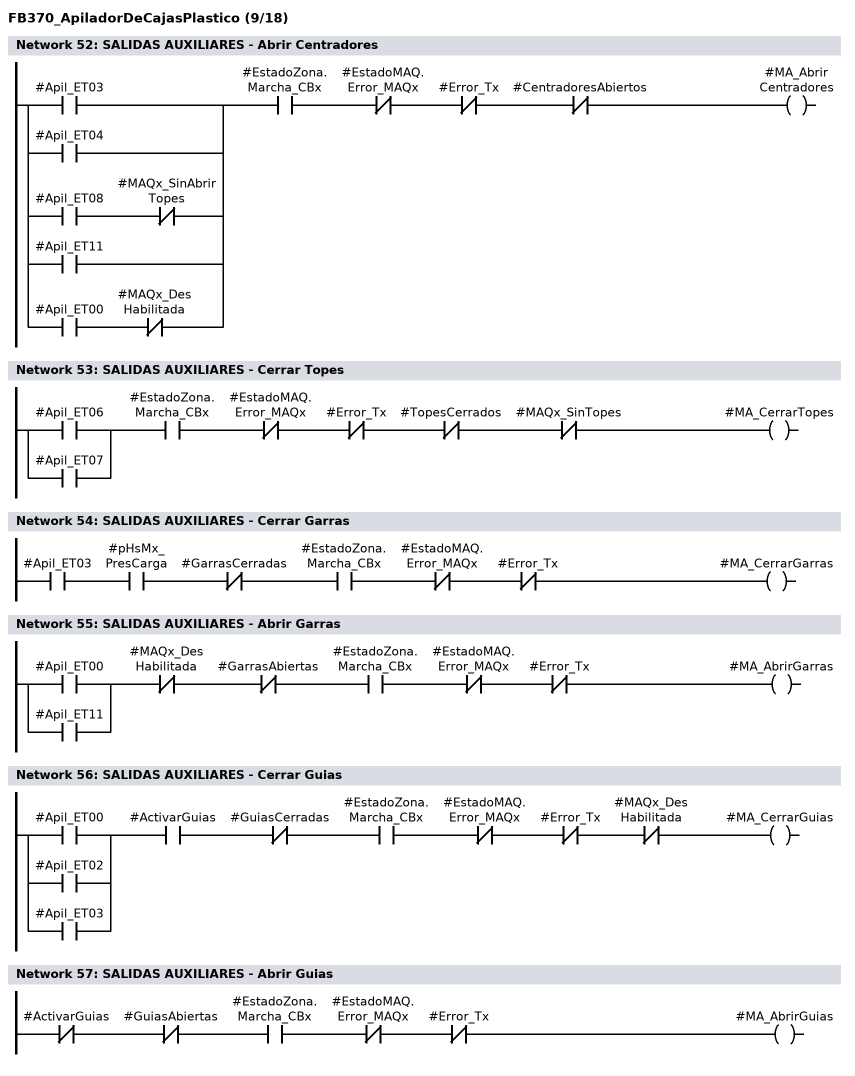
   RUNG wire#powerrail
      Contact( #Apil_ET03 )
      wire#w1
      Contact( #EstadoZona.Marcha_CBx )
      I_Contact( #EstadoMAQ.Error_MAQx )
      I_Contact( #Error_Tx )
      I_Contact( #CentradoresAbiertos )
      Coil( #MA_AbrirCentradores )
   END_RUNG
   RUNG wire#powerrail
      Contact( #Apil_ET04 )
   END_RUNG wire#w1
   RUNG wire#powerrail
      Contact( #Apil_ET08 )
      I_Contact( #MAQx_SinAbrirTopes )
   END_RUNG wire#w1
   RUNG wire#powerrail
      Contact( #Apil_ET11 )
   END_RUNG wire#w1
   RUNG wire#powerrail
      Contact( #Apil_ET00 )
      I_Contact( #MAQx_DesHabilitada )
   END_RUNG wire#w1
   // the same network as SCL:
   #MA_AbrirCentradores := (#Apil_ET03 OR #Apil_ET04 OR (#Apil_ET08 AND NOT #MAQx_SinAbrirTopes) OR #Apil_ET11 OR (#Apil_ET00 AND NOT #MAQx_DesHabilitada)) AND #EstadoZona.Marcha_CBx AND NOT #EstadoMAQ.Error_MAQx AND NOT #Error_Tx AND NOT #CentradoresAbiertos;
END_REGION

REGION Network 53: SALIDAS AUXILIARES - Cerrar Topes
   RUNG wire#powerrail
      Contact( #Apil_ET06 )
      wire#w1
      Contact( #EstadoZona.Marcha_CBx )
      I_Contact( #EstadoMAQ.Error_MAQx )
      I_Contact( #Error_Tx )
      I_Contact( #TopesCerrados )
      I_Contact( #MAQx_SinTopes )
      Coil( #MA_CerrarTopes )
   END_RUNG
   RUNG wire#powerrail
      Contact( #Apil_ET07 )
   END_RUNG wire#w1
   // the same network as SCL:
   #MA_CerrarTopes := (#Apil_ET06 OR #Apil_ET07) AND #EstadoZona.Marcha_CBx AND NOT #EstadoMAQ.Error_MAQx AND NOT #Error_Tx AND NOT #TopesCerrados AND NOT #MAQx_SinTopes;
END_REGION

REGION Network 54: SALIDAS AUXILIARES - Cerrar Garras
   RUNG wire#powerrail
      Contact( #Apil_ET03 )
      Contact( #pHsMx_PresCarga )
      I_Contact( #GarrasCerradas )
      Contact( #EstadoZona.Marcha_CBx )
      I_Contact( #EstadoMAQ.Error_MAQx )
      I_Contact( #Error_Tx )
      Coil( #MA_CerrarGarras )
   END_RUNG
   // the same network as SCL:
   #MA_CerrarGarras := #Apil_ET03 AND #pHsMx_PresCarga AND NOT #GarrasCerradas AND #EstadoZona.Marcha_CBx AND NOT #EstadoMAQ.Error_MAQx AND NOT #Error_Tx;
END_REGION

REGION Network 55: SALIDAS AUXILIARES - Abrir Garras
   RUNG wire#powerrail
      Contact( #Apil_ET00 )
      wire#w1
      I_Contact( #MAQx_DesHabilitada )
      I_Contact( #GarrasAbiertas )
      Contact( #EstadoZona.Marcha_CBx )
      I_Contact( #EstadoMAQ.Error_MAQx )
      I_Contact( #Error_Tx )
      Coil( #MA_AbrirGarras )
   END_RUNG
   RUNG wire#powerrail
      Contact( #Apil_ET11 )
   END_RUNG wire#w1
   // the same network as SCL:
   #MA_AbrirGarras := (#Apil_ET00 OR #Apil_ET11) AND NOT #MAQx_DesHabilitada AND NOT #GarrasAbiertas AND #EstadoZona.Marcha_CBx AND NOT #EstadoMAQ.Error_MAQx AND NOT #Error_Tx;
END_REGION

REGION Network 56: SALIDAS AUXILIARES - Cerrar Guias
   RUNG wire#powerrail
      Contact( #Apil_ET00 )
      wire#w1
      Contact( #ActivarGuias )
      I_Contact( #GuiasCerradas )
      Contact( #EstadoZona.Marcha_CBx )
      I_Contact( #EstadoMAQ.Error_MAQx )
      I_Contact( #Error_Tx )
      I_Contact( #MAQx_DesHabilitada )
      Coil( #MA_CerrarGuias )
   END_RUNG
   RUNG wire#powerrail
      Contact( #Apil_ET02 )
   END_RUNG wire#w1
   RUNG wire#powerrail
      Contact( #Apil_ET03 )
   END_RUNG wire#w1
   // the same network as SCL:
   #MA_CerrarGuias := (#Apil_ET00 OR #Apil_ET02 OR #Apil_ET03) AND #ActivarGuias AND NOT #GuiasCerradas AND #EstadoZona.Marcha_CBx AND NOT #EstadoMAQ.Error_MAQx AND NOT #Error_Tx AND NOT #MAQx_DesHabilitada;
END_REGION

REGION Network 57: SALIDAS AUXILIARES - Abrir Guias
   RUNG wire#powerrail
      I_Contact( #ActivarGuias )
      I_Contact( #GuiasAbiertas )
      Contact( #EstadoZona.Marcha_CBx )
      I_Contact( #EstadoMAQ.Error_MAQx )
      I_Contact( #Error_Tx )
      Coil( #MA_AbrirGuias )
   END_RUNG
   // the same network as SCL:
   #MA_AbrirGuias := NOT #ActivarGuias AND NOT #GuiasAbiertas AND #EstadoZona.Marcha_CBx AND NOT #EstadoMAQ.Error_MAQx AND NOT #Error_Tx;
END_REGION

REGION Network 58: SALIDAS EXTERIORES - CONTROL DE CENTRADOR CF1CF2 - Abrir y Cerrar >>> Tope de Caja Grande
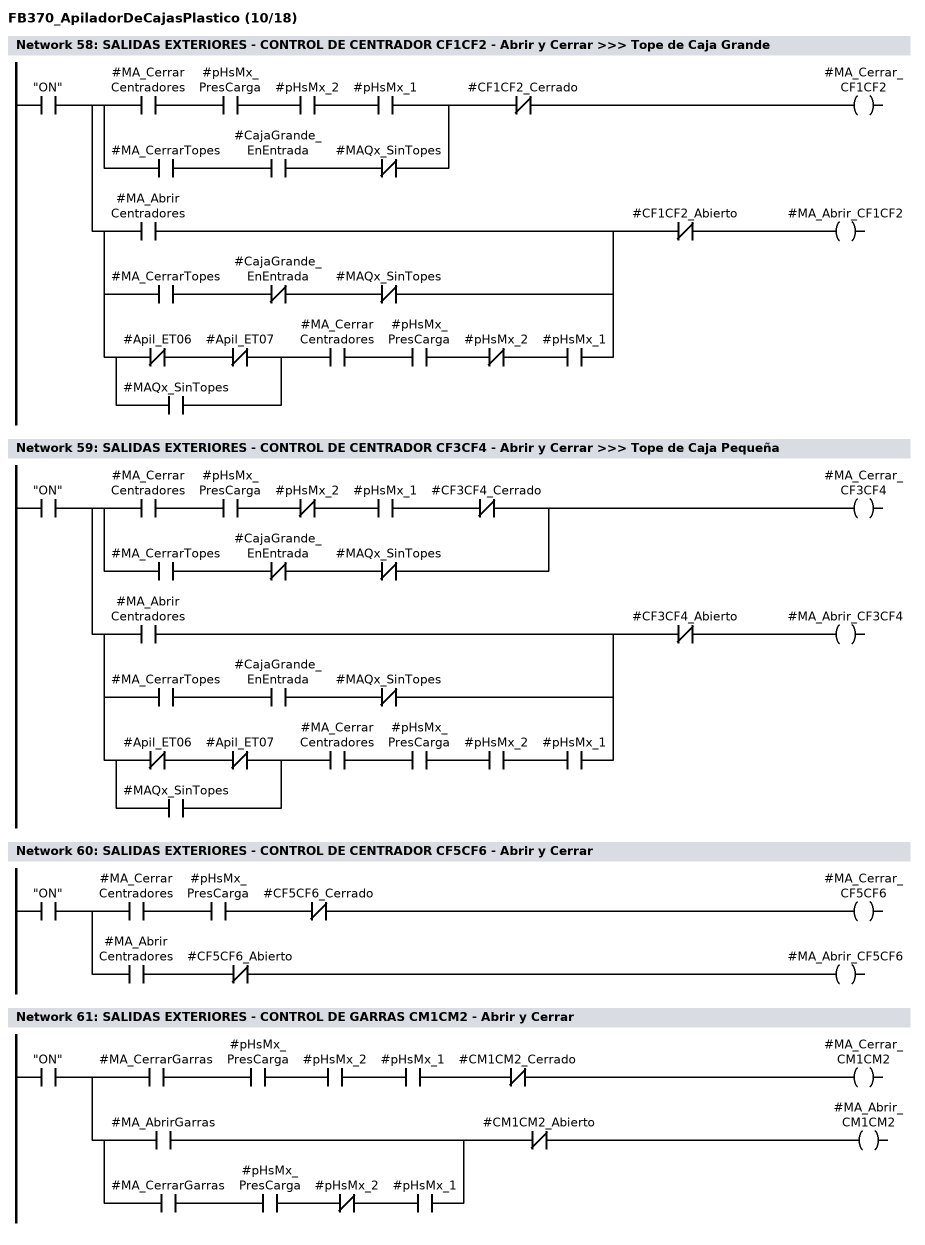
   RUNG wire#powerrail
      Contact( "ON" )
      wire#w1
      Contact( #MA_CerrarCentradores )
      Contact( #pHsMx_PresCarga )
      Contact( #pHsMx_2 )
      Contact( #pHsMx_1 )
      wire#w2
      I_Contact( #CF1CF2_Cerrado )
      Coil( #MA_Cerrar_CF1CF2 )
   END_RUNG
   RUNG wire#w1
      Contact( #MA_CerrarTopes )
      Contact( #CajaGrande_EnEntrada )
      I_Contact( #MAQx_SinTopes )
   END_RUNG wire#w2
   RUNG wire#w1
      Contact( #MA_AbrirCentradores )
      wire#w3
      I_Contact( #CF1CF2_Abierto )
      Coil( #MA_Abrir_CF1CF2 )
   END_RUNG
   RUNG wire#w1
      Contact( #MA_CerrarTopes )
      I_Contact( #CajaGrande_EnEntrada )
      I_Contact( #MAQx_SinTopes )
   END_RUNG wire#w3
   RUNG wire#w1
      I_Contact( #Apil_ET06 )
      I_Contact( #Apil_ET07 )
      wire#w4
      Contact( #MA_CerrarCentradores )
      Contact( #pHsMx_PresCarga )
      I_Contact( #pHsMx_2 )
      Contact( #pHsMx_1 )
   END_RUNG wire#w3
   RUNG wire#w1
      Contact( #MAQx_SinTopes )
   END_RUNG wire#w4
   // the same network as SCL:
   #MA_Cerrar_CF1CF2 := "ON" AND ((#MA_CerrarCentradores AND #pHsMx_PresCarga AND #pHsMx_2 AND #pHsMx_1) OR (#MA_CerrarTopes AND #CajaGrande_EnEntrada AND NOT #MAQx_SinTopes)) AND NOT #CF1CF2_Cerrado;
   #MA_Abrir_CF1CF2 := "ON" AND (#MA_AbrirCentradores OR (#MA_CerrarTopes AND NOT #CajaGrande_EnEntrada AND NOT #MAQx_SinTopes) OR (((NOT #Apil_ET06 AND NOT #Apil_ET07) OR #MAQx_SinTopes) AND #MA_CerrarCentradores AND #pHsMx_PresCarga AND NOT #pHsMx_2 AND #pHsMx_1)) AND NOT #CF1CF2_Abierto;
END_REGION

REGION Network 59: SALIDAS EXTERIORES - CONTROL DE CENTRADOR CF3CF4 - Abrir y Cerrar >>> Tope de Caja Pequeña
   RUNG wire#powerrail
      Contact( "ON" )
      wire#w1
      Contact( #MA_CerrarCentradores )
      Contact( #pHsMx_PresCarga )
      I_Contact( #pHsMx_2 )
      Contact( #pHsMx_1 )
      I_Contact( #CF3CF4_Cerrado )
      wire#w2
      Coil( #MA_Cerrar_CF3CF4 )
   END_RUNG
   RUNG wire#w1
      Contact( #MA_CerrarTopes )
      I_Contact( #CajaGrande_EnEntrada )
      I_Contact( #MAQx_SinTopes )
   END_RUNG wire#w2
   RUNG wire#w1
      Contact( #MA_AbrirCentradores )
      wire#w3
      I_Contact( #CF3CF4_Abierto )
      Coil( #MA_Abrir_CF3CF4 )
   END_RUNG
   RUNG wire#w1
      Contact( #MA_CerrarTopes )
      Contact( #CajaGrande_EnEntrada )
      I_Contact( #MAQx_SinTopes )
   END_RUNG wire#w3
   RUNG wire#w1
      I_Contact( #Apil_ET06 )
      I_Contact( #Apil_ET07 )
      wire#w4
      Contact( #MA_CerrarCentradores )
      Contact( #pHsMx_PresCarga )
      Contact( #pHsMx_2 )
      Contact( #pHsMx_1 )
   END_RUNG wire#w3
   RUNG wire#w1
      Contact( #MAQx_SinTopes )
   END_RUNG wire#w4
   // the same network as SCL:
   #MA_Cerrar_CF3CF4 := "ON" AND ((#MA_CerrarCentradores AND #pHsMx_PresCarga AND NOT #pHsMx_2 AND #pHsMx_1 AND NOT #CF3CF4_Cerrado) OR (#MA_CerrarTopes AND NOT #CajaGrande_EnEntrada AND NOT #MAQx_SinTopes));
   #MA_Abrir_CF3CF4 := "ON" AND (#MA_AbrirCentradores OR (#MA_CerrarTopes AND #CajaGrande_EnEntrada AND NOT #MAQx_SinTopes) OR (((NOT #Apil_ET06 AND NOT #Apil_ET07) OR #MAQx_SinTopes) AND #MA_CerrarCentradores AND #pHsMx_PresCarga AND #pHsMx_2 AND #pHsMx_1)) AND NOT #CF3CF4_Abierto;
END_REGION

REGION Network 60: SALIDAS EXTERIORES - CONTROL DE CENTRADOR CF5CF6 - Abrir y Cerrar
   RUNG wire#powerrail
      Contact( "ON" )
      wire#w1
      Contact( #MA_CerrarCentradores )
      Contact( #pHsMx_PresCarga )
      I_Contact( #CF5CF6_Cerrado )
      Coil( #MA_Cerrar_CF5CF6 )
   END_RUNG
   RUNG wire#w1
      Contact( #MA_AbrirCentradores )
      I_Contact( #CF5CF6_Abierto )
      Coil( #MA_Abrir_CF5CF6 )
   END_RUNG
   // the same network as SCL:
   #MA_Cerrar_CF5CF6 := "ON" AND #MA_CerrarCentradores AND #pHsMx_PresCarga AND NOT #CF5CF6_Cerrado;
   #MA_Abrir_CF5CF6 := "ON" AND #MA_AbrirCentradores AND NOT #CF5CF6_Abierto;
END_REGION

REGION Network 61: SALIDAS EXTERIORES - CONTROL DE GARRAS CM1CM2 - Abrir y Cerrar
   RUNG wire#powerrail
      Contact( "ON" )
      wire#w1
      Contact( #MA_CerrarGarras )
      Contact( #pHsMx_PresCarga )
      Contact( #pHsMx_2 )
      Contact( #pHsMx_1 )
      I_Contact( #CM1CM2_Cerrado )
      Coil( #MA_Cerrar_CM1CM2 )
   END_RUNG
   RUNG wire#w1
      Contact( #MA_AbrirGarras )
      wire#w2
      I_Contact( #CM1CM2_Abierto )
      Coil( #MA_Abrir_CM1CM2 )
   END_RUNG
   RUNG wire#w1
      Contact( #MA_CerrarGarras )
      Contact( #pHsMx_PresCarga )
      I_Contact( #pHsMx_2 )
      Contact( #pHsMx_1 )
   END_RUNG wire#w2
   // the same network as SCL:
   #MA_Cerrar_CM1CM2 := "ON" AND #MA_CerrarGarras AND #pHsMx_PresCarga AND #pHsMx_2 AND #pHsMx_1 AND NOT #CM1CM2_Cerrado;
   #MA_Abrir_CM1CM2 := "ON" AND (#MA_AbrirGarras OR (#MA_CerrarGarras AND #pHsMx_PresCarga AND NOT #pHsMx_2 AND #pHsMx_1)) AND NOT #CM1CM2_Abierto;
END_REGION

REGION Network 62: SALIDAS EXTERIORES - CONTROL DE GARRAS CM3CM4 - Abrir y Cerrar >>> Caja EuroPool CM3CM8
   // Nota: Caja Tipo Europool >>> Utilizar para Caja Pequeña
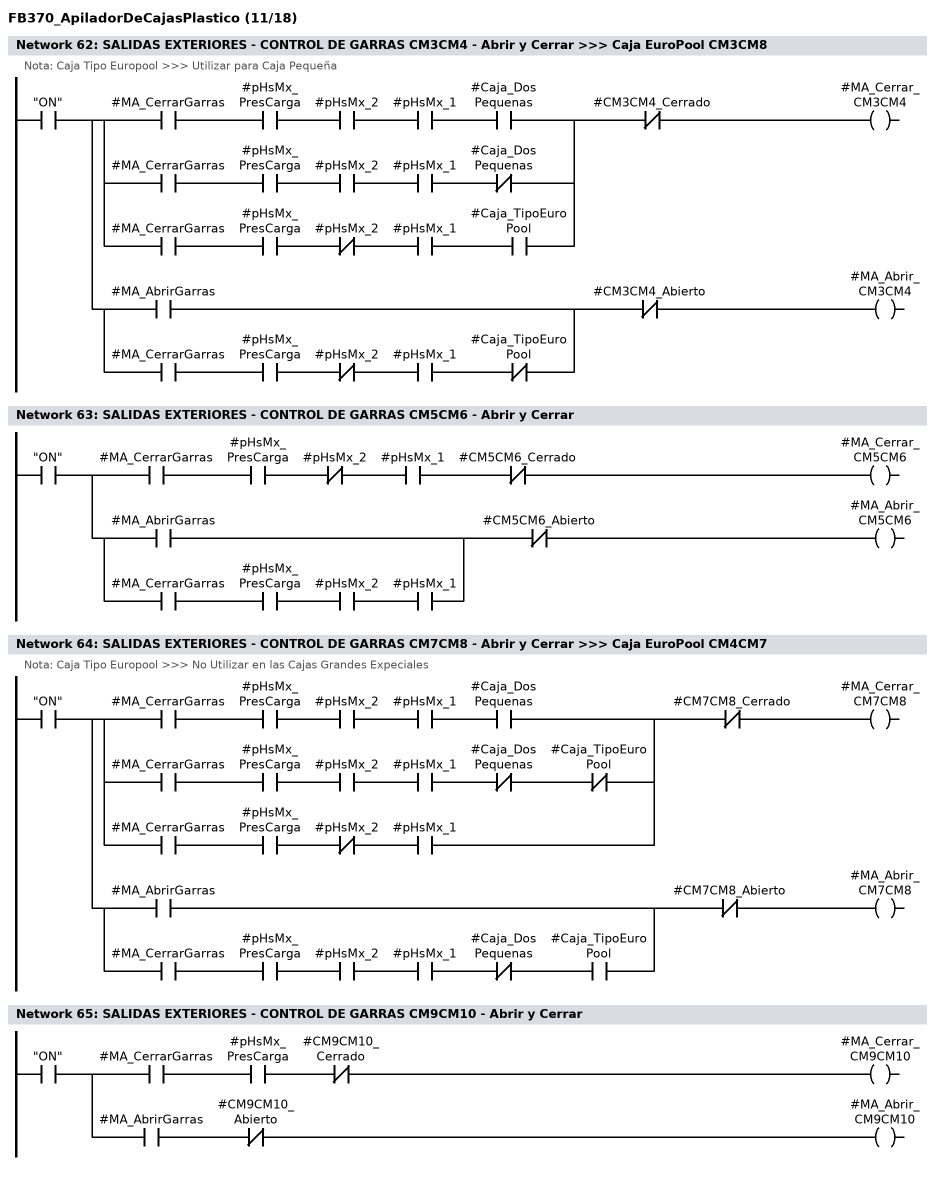
   RUNG wire#powerrail
      Contact( "ON" )
      wire#w1
      Contact( #MA_CerrarGarras )
      Contact( #pHsMx_PresCarga )
      Contact( #pHsMx_2 )
      Contact( #pHsMx_1 )
      Contact( #Caja_DosPequenas )
      wire#w2
      I_Contact( #CM3CM4_Cerrado )
      Coil( #MA_Cerrar_CM3CM4 )
   END_RUNG
   RUNG wire#w1
      Contact( #MA_CerrarGarras )
      Contact( #pHsMx_PresCarga )
      Contact( #pHsMx_2 )
      Contact( #pHsMx_1 )
      I_Contact( #Caja_DosPequenas )
   END_RUNG wire#w2
   RUNG wire#w1
      Contact( #MA_CerrarGarras )
      Contact( #pHsMx_PresCarga )
      I_Contact( #pHsMx_2 )
      Contact( #pHsMx_1 )
      Contact( #Caja_TipoEuroPool )
   END_RUNG wire#w2
   RUNG wire#w1
      Contact( #MA_AbrirGarras )
      wire#w3
      I_Contact( #CM3CM4_Abierto )
      Coil( #MA_Abrir_CM3CM4 )
   END_RUNG
   RUNG wire#w1
      Contact( #MA_CerrarGarras )
      Contact( #pHsMx_PresCarga )
      I_Contact( #pHsMx_2 )
      Contact( #pHsMx_1 )
      I_Contact( #Caja_TipoEuroPool )
   END_RUNG wire#w3
   // the same network as SCL:
   #MA_Cerrar_CM3CM4 := "ON" AND ((#MA_CerrarGarras AND #pHsMx_PresCarga AND #pHsMx_2 AND #pHsMx_1 AND #Caja_DosPequenas) OR (#MA_CerrarGarras AND #pHsMx_PresCarga AND #pHsMx_2 AND #pHsMx_1 AND NOT #Caja_DosPequenas) OR (#MA_CerrarGarras AND #pHsMx_PresCarga AND NOT #pHsMx_2 AND #pHsMx_1 AND #Caja_TipoEuroPool)) AND NOT #CM3CM4_Cerrado;
   #MA_Abrir_CM3CM4 := "ON" AND (#MA_AbrirGarras OR (#MA_CerrarGarras AND #pHsMx_PresCarga AND NOT #pHsMx_2 AND #pHsMx_1 AND NOT #Caja_TipoEuroPool)) AND NOT #CM3CM4_Abierto;
END_REGION

REGION Network 63: SALIDAS EXTERIORES - CONTROL DE GARRAS CM5CM6 - Abrir y Cerrar
   RUNG wire#powerrail
      Contact( "ON" )
      wire#w1
      Contact( #MA_CerrarGarras )
      Contact( #pHsMx_PresCarga )
      I_Contact( #pHsMx_2 )
      Contact( #pHsMx_1 )
      I_Contact( #CM5CM6_Cerrado )
      Coil( #MA_Cerrar_CM5CM6 )
   END_RUNG
   RUNG wire#w1
      Contact( #MA_AbrirGarras )
      wire#w2
      I_Contact( #CM5CM6_Abierto )
      Coil( #MA_Abrir_CM5CM6 )
   END_RUNG
   RUNG wire#w1
      Contact( #MA_CerrarGarras )
      Contact( #pHsMx_PresCarga )
      Contact( #pHsMx_2 )
      Contact( #pHsMx_1 )
   END_RUNG wire#w2
   // the same network as SCL:
   #MA_Cerrar_CM5CM6 := "ON" AND #MA_CerrarGarras AND #pHsMx_PresCarga AND NOT #pHsMx_2 AND #pHsMx_1 AND NOT #CM5CM6_Cerrado;
   #MA_Abrir_CM5CM6 := "ON" AND (#MA_AbrirGarras OR (#MA_CerrarGarras AND #pHsMx_PresCarga AND #pHsMx_2 AND #pHsMx_1)) AND NOT #CM5CM6_Abierto;
END_REGION

REGION Network 64: SALIDAS EXTERIORES - CONTROL DE GARRAS CM7CM8 - Abrir y Cerrar >>> Caja EuroPool CM4CM7
   // Nota: Caja Tipo Europool >>> No Utilizar en las Cajas Grandes Expeciales
   RUNG wire#powerrail
      Contact( "ON" )
      wire#w1
      Contact( #MA_CerrarGarras )
      Contact( #pHsMx_PresCarga )
      Contact( #pHsMx_2 )
      Contact( #pHsMx_1 )
      Contact( #Caja_DosPequenas )
      wire#w2
      I_Contact( #CM7CM8_Cerrado )
      Coil( #MA_Cerrar_CM7CM8 )
   END_RUNG
   RUNG wire#w1
      Contact( #MA_CerrarGarras )
      Contact( #pHsMx_PresCarga )
      Contact( #pHsMx_2 )
      Contact( #pHsMx_1 )
      I_Contact( #Caja_DosPequenas )
      I_Contact( #Caja_TipoEuroPool )
   END_RUNG wire#w2
   RUNG wire#w1
      Contact( #MA_CerrarGarras )
      Contact( #pHsMx_PresCarga )
      I_Contact( #pHsMx_2 )
      Contact( #pHsMx_1 )
   END_RUNG wire#w2
   RUNG wire#w1
      Contact( #MA_AbrirGarras )
      wire#w3
      I_Contact( #CM7CM8_Abierto )
      Coil( #MA_Abrir_CM7CM8 )
   END_RUNG
   RUNG wire#w1
      Contact( #MA_CerrarGarras )
      Contact( #pHsMx_PresCarga )
      Contact( #pHsMx_2 )
      Contact( #pHsMx_1 )
      I_Contact( #Caja_DosPequenas )
      Contact( #Caja_TipoEuroPool )
   END_RUNG wire#w3
   // the same network as SCL:
   #MA_Cerrar_CM7CM8 := "ON" AND ((#MA_CerrarGarras AND #pHsMx_PresCarga AND #pHsMx_2 AND #pHsMx_1 AND #Caja_DosPequenas) OR (#MA_CerrarGarras AND #pHsMx_PresCarga AND #pHsMx_2 AND #pHsMx_1 AND NOT #Caja_DosPequenas AND NOT #Caja_TipoEuroPool) OR (#MA_CerrarGarras AND #pHsMx_PresCarga AND NOT #pHsMx_2 AND #pHsMx_1)) AND NOT #CM7CM8_Cerrado;
   #MA_Abrir_CM7CM8 := "ON" AND (#MA_AbrirGarras OR (#MA_CerrarGarras AND #pHsMx_PresCarga AND #pHsMx_2 AND #pHsMx_1 AND NOT #Caja_DosPequenas AND #Caja_TipoEuroPool)) AND NOT #CM7CM8_Abierto;
END_REGION

REGION Network 65: SALIDAS EXTERIORES - CONTROL DE GARRAS CM9CM10 - Abrir y Cerrar
   RUNG wire#powerrail
      Contact( "ON" )
      wire#w1
      Contact( #MA_CerrarGarras )
      Contact( #pHsMx_PresCarga )
      I_Contact( #CM9CM10_Cerrado )
      Coil( #MA_Cerrar_CM9CM10 )
   END_RUNG
   RUNG wire#w1
      Contact( #MA_AbrirGarras )
      I_Contact( #CM9CM10_Abierto )
      Coil( #MA_Abrir_CM9CM10 )
   END_RUNG
   // the same network as SCL:
   #MA_Cerrar_CM9CM10 := "ON" AND #MA_CerrarGarras AND #pHsMx_PresCarga AND NOT #CM9CM10_Cerrado;
   #MA_Abrir_CM9CM10 := "ON" AND #MA_AbrirGarras AND NOT #CM9CM10_Abierto;
END_REGION

REGION Network 66: SALIDAS EXTERIORES - CONTROL DE GUIAS GF1GF2 - Abrir y Cerrar
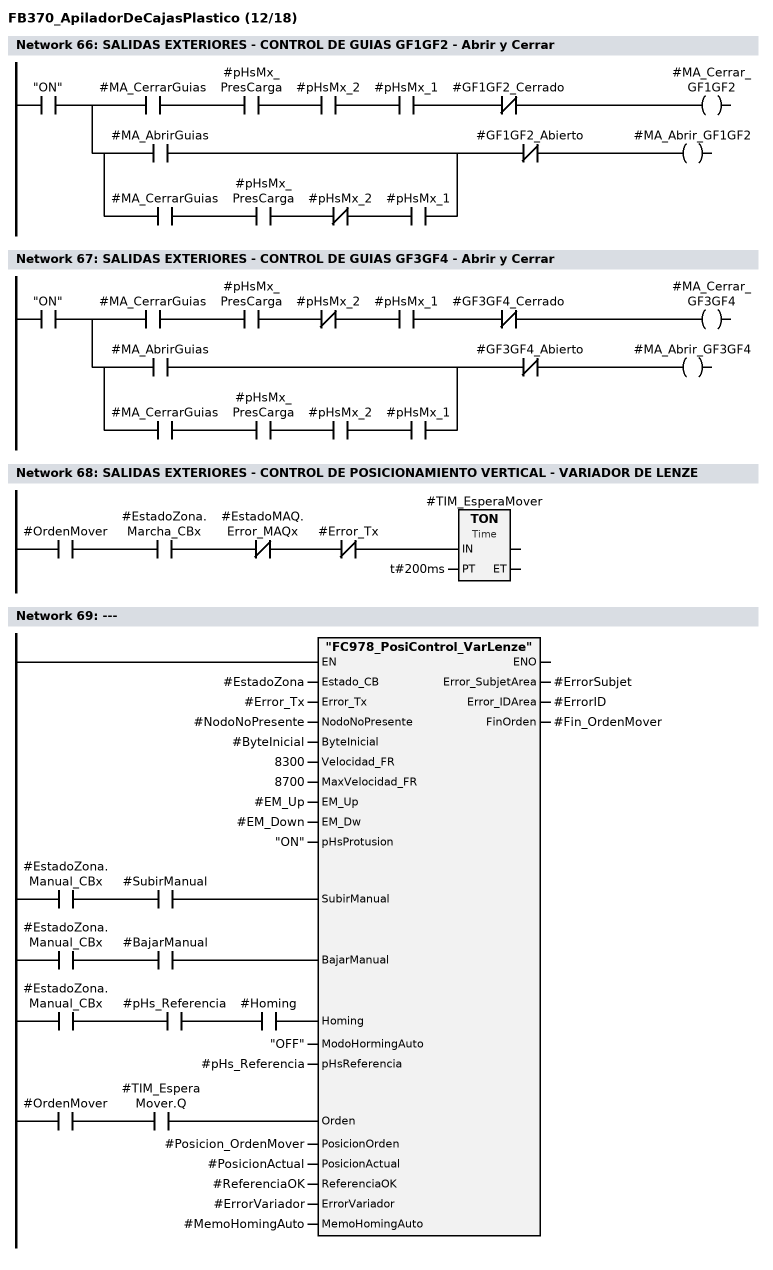
   RUNG wire#powerrail
      Contact( "ON" )
      wire#w1
      Contact( #MA_CerrarGuias )
      Contact( #pHsMx_PresCarga )
      Contact( #pHsMx_2 )
      Contact( #pHsMx_1 )
      I_Contact( #GF1GF2_Cerrado )
      Coil( #MA_Cerrar_GF1GF2 )
   END_RUNG
   RUNG wire#w1
      Contact( #MA_AbrirGuias )
      wire#w2
      I_Contact( #GF1GF2_Abierto )
      Coil( #MA_Abrir_GF1GF2 )
   END_RUNG
   RUNG wire#w1
      Contact( #MA_CerrarGuias )
      Contact( #pHsMx_PresCarga )
      I_Contact( #pHsMx_2 )
      Contact( #pHsMx_1 )
   END_RUNG wire#w2
   // the same network as SCL:
   #MA_Cerrar_GF1GF2 := "ON" AND #MA_CerrarGuias AND #pHsMx_PresCarga AND #pHsMx_2 AND #pHsMx_1 AND NOT #GF1GF2_Cerrado;
   #MA_Abrir_GF1GF2 := "ON" AND (#MA_AbrirGuias OR (#MA_CerrarGuias AND #pHsMx_PresCarga AND NOT #pHsMx_2 AND #pHsMx_1)) AND NOT #GF1GF2_Abierto;
END_REGION

REGION Network 67: SALIDAS EXTERIORES - CONTROL DE GUIAS GF3GF4 - Abrir y Cerrar
   RUNG wire#powerrail
      Contact( "ON" )
      wire#w1
      Contact( #MA_CerrarGuias )
      Contact( #pHsMx_PresCarga )
      I_Contact( #pHsMx_2 )
      Contact( #pHsMx_1 )
      I_Contact( #GF3GF4_Cerrado )
      Coil( #MA_Cerrar_GF3GF4 )
   END_RUNG
   RUNG wire#w1
      Contact( #MA_AbrirGuias )
      wire#w2
      I_Contact( #GF3GF4_Abierto )
      Coil( #MA_Abrir_GF3GF4 )
   END_RUNG
   RUNG wire#w1
      Contact( #MA_CerrarGuias )
      Contact( #pHsMx_PresCarga )
      Contact( #pHsMx_2 )
      Contact( #pHsMx_1 )
   END_RUNG wire#w2
   // the same network as SCL:
   #MA_Cerrar_GF3GF4 := "ON" AND #MA_CerrarGuias AND #pHsMx_PresCarga AND NOT #pHsMx_2 AND #pHsMx_1 AND NOT #GF3GF4_Cerrado;
   #MA_Abrir_GF3GF4 := "ON" AND (#MA_AbrirGuias OR (#MA_CerrarGuias AND #pHsMx_PresCarga AND #pHsMx_2 AND #pHsMx_1)) AND NOT #GF3GF4_Abierto;
END_REGION

REGION Network 68: SALIDAS EXTERIORES - CONTROL DE POSICIONAMIENTO VERTICAL - VARIADOR DE LENZE
   RUNG wire#powerrail
      Contact( #OrdenMover )
      Contact( #EstadoZona.Marcha_CBx )
      I_Contact( #EstadoMAQ.Error_MAQx )
      I_Contact( #Error_Tx )
      { S7_Templates := "time_type := Time" } #TIM_EsperaMover.TON(pt := t#200ms, et =>)
   END_RUNG
   // the same network as SCL:
   #TIM_EsperaMover(IN := #OrdenMover AND #EstadoZona.Marcha_CBx AND NOT #EstadoMAQ.Error_MAQx AND NOT #Error_Tx,   // TON
                    PT := t#200ms);
END_REGION

REGION Network 69: ---
   RUNG wire#powerrail
      "FC978_PosiControl_VarLenze"(SubirManual := wire#w1, BajarManual := wire#w2, Homing := wire#w3, Orden := wire#w4, Estado_CB := #EstadoZona, Error_Tx := #Error_Tx, NodoNoPresente := #NodoNoPresente, ByteInicial := #ByteInicial, Velocidad_FR := 8300, MaxVelocidad_FR := 8700, EM_Up := #EM_Up, EM_Dw := #EM_Down, pHsProtusion := "ON", ModoHormingAuto := "OFF", pHsReferencia := #pHs_Referencia, PosicionOrden := #Posicion_OrdenMover, PosicionActual := #PosicionActual, ReferenciaOK := #ReferenciaOK, ErrorVariador := #ErrorVariador, MemoHomingAuto := #MemoHomingAuto, Error_SubjetArea => #ErrorSubjet, Error_IDArea => #ErrorID, FinOrden => #Fin_OrdenMover)
   END_RUNG
   RUNG wire#powerrail
      Contact( #EstadoZona.Manual_CBx )
      Contact( #SubirManual )
   END_RUNG wire#w1
   RUNG wire#powerrail
      Contact( #EstadoZona.Manual_CBx )
      Contact( #BajarManual )
   END_RUNG wire#w2
   RUNG wire#powerrail
      Contact( #EstadoZona.Manual_CBx )
      Contact( #pHs_Referencia )
      Contact( #Homing )
   END_RUNG wire#w3
   RUNG wire#powerrail
      Contact( #OrdenMover )
      Contact( #TIM_EsperaMover.Q )
   END_RUNG wire#w4
   // the same network as SCL:
   "FC978_PosiControl_VarLenze"(Estado_CB := #EstadoZona,
                           Error_Tx := #Error_Tx,
                           NodoNoPresente := #NodoNoPresente,
                           ByteInicial := #ByteInicial,
                           Velocidad_FR := 8300,
                           MaxVelocidad_FR := 8700,
                           EM_Up := #EM_Up,
                           EM_Dw := #EM_Down,
                           pHsProtusion := "ON",
                           SubirManual := #EstadoZona.Manual_CBx AND #SubirManual,
                           BajarManual := #EstadoZona.Manual_CBx AND #BajarManual,
                           Homing := #EstadoZona.Manual_CBx AND #pHs_Referencia AND #Homing,
                           ModoHormingAuto := "OFF",
                           pHsReferencia := #pHs_Referencia,
                           Orden := #OrdenMover AND #TIM_EsperaMover.Q,
                           PosicionOrden := #Posicion_OrdenMover,
                           PosicionActual := #PosicionActual,
                           ReferenciaOK := #ReferenciaOK,
                           ErrorVariador := #ErrorVariador,
                           MemoHomingAuto := #MemoHomingAuto,
                           Error_SubjetArea => #ErrorSubjet,
                           Error_IDArea => #ErrorID,
                           FinOrden => #Fin_OrdenMover);
END_REGION

REGION Network 70: TMP - Espera En Tension
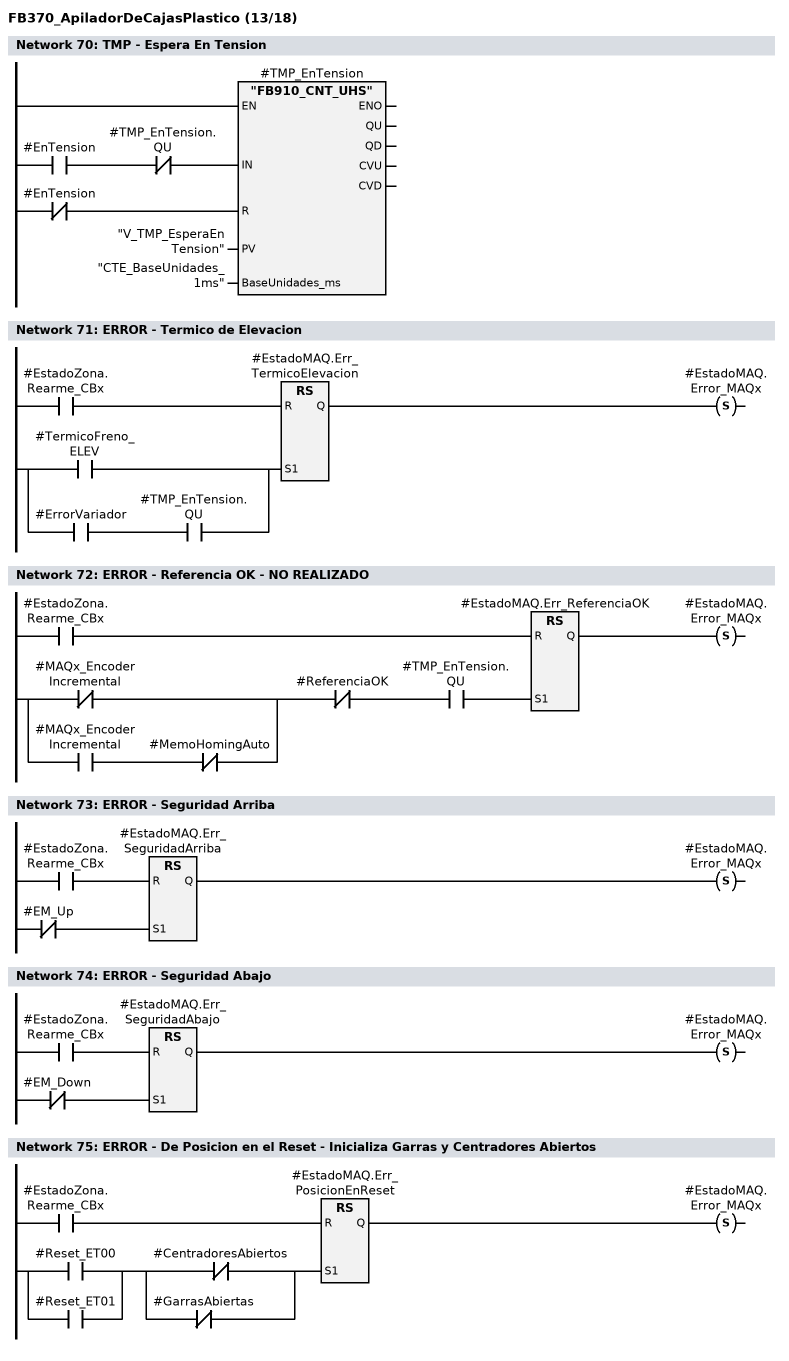
   RUNG wire#powerrail
      #TMP_EnTension(IN := wire#w1, R := wire#w2, PV := "V_TMP_EsperaEnTension", BaseUnidades_ms := "CTE_BaseUnidades_1ms", QU =>, QD =>, CVU =>, CVD =>)
   END_RUNG
   RUNG wire#powerrail
      Contact( #EnTension )
      I_Contact( #TMP_EnTension.QU )
   END_RUNG wire#w1
   RUNG wire#powerrail
      I_Contact( #EnTension )
   END_RUNG wire#w2
   // the same network as SCL:
   #TMP_EnTension(IN := #EnTension AND NOT #TMP_EnTension.QU,   // "FB910_CNT_UHS"
                  R := NOT #EnTension,
                  PV := "V_TMP_EsperaEnTension",
                  BaseUnidades_ms := "CTE_BaseUnidades_1ms");
END_REGION

REGION Network 71: ERROR - Termico de Elevacion
   RUNG wire#powerrail
      Contact( #EstadoZona.Rearme_CBx )
      S_RS(operand := #EstadoMAQ.Err_TermicoElevacion, s1 := wire#w1)
      S_Coil( #EstadoMAQ.Error_MAQx )
   END_RUNG
   RUNG wire#powerrail
      Contact( #TermicoFreno_ELEV )
   END_RUNG wire#w1
   RUNG wire#powerrail
      Contact( #ErrorVariador )
      Contact( #TMP_EnTension.QU )
   END_RUNG wire#w1
   // the same network as SCL:
   IF #EstadoZona.Rearme_CBx THEN
       #EstadoMAQ.Err_TermicoElevacion := FALSE;   // RS flip-flop
   END_IF;
   IF #TermicoFreno_ELEV OR (#ErrorVariador AND #TMP_EnTension.QU) THEN
       #EstadoMAQ.Err_TermicoElevacion := TRUE;
   END_IF;
   IF #EstadoMAQ.Err_TermicoElevacion THEN #EstadoMAQ.Error_MAQx := TRUE; END_IF;
END_REGION

REGION Network 72: ERROR - Referencia OK - NO REALIZADO
   RUNG wire#powerrail
      Contact( #EstadoZona.Rearme_CBx )
      S_RS(operand := #EstadoMAQ.Err_ReferenciaOK, s1 := wire#w2)
      S_Coil( #EstadoMAQ.Error_MAQx )
   END_RUNG
   RUNG wire#powerrail
      I_Contact( #MAQx_EncoderIncremental )
      wire#w1
      I_Contact( #ReferenciaOK )
      Contact( #TMP_EnTension.QU )
   END_RUNG wire#w2
   RUNG wire#powerrail
      Contact( #MAQx_EncoderIncremental )
      I_Contact( #MemoHomingAuto )
   END_RUNG wire#w1
   // the same network as SCL:
   IF #EstadoZona.Rearme_CBx THEN
       #EstadoMAQ.Err_ReferenciaOK := FALSE;   // RS flip-flop
   END_IF;
   IF (NOT #MAQx_EncoderIncremental OR (#MAQx_EncoderIncremental AND NOT #MemoHomingAuto)) AND NOT #ReferenciaOK AND #TMP_EnTension.QU THEN
       #EstadoMAQ.Err_ReferenciaOK := TRUE;
   END_IF;
   IF #EstadoMAQ.Err_ReferenciaOK THEN #EstadoMAQ.Error_MAQx := TRUE; END_IF;
END_REGION

REGION Network 73: ERROR - Seguridad Arriba
   RUNG wire#powerrail
      Contact( #EstadoZona.Rearme_CBx )
      S_RS(operand := #EstadoMAQ.Err_SeguridadArriba, s1 := wire#w1)
      S_Coil( #EstadoMAQ.Error_MAQx )
   END_RUNG
   RUNG wire#powerrail
      I_Contact( #EM_Up )
   END_RUNG wire#w1
   // the same network as SCL:
   IF #EstadoZona.Rearme_CBx THEN
       #EstadoMAQ.Err_SeguridadArriba := FALSE;   // RS flip-flop
   END_IF;
   IF NOT #EM_Up THEN #EstadoMAQ.Err_SeguridadArriba := TRUE; END_IF;
   IF #EstadoMAQ.Err_SeguridadArriba THEN #EstadoMAQ.Error_MAQx := TRUE; END_IF;
END_REGION

REGION Network 74: ERROR - Seguridad Abajo
   RUNG wire#powerrail
      Contact( #EstadoZona.Rearme_CBx )
      S_RS(operand := #EstadoMAQ.Err_SeguridadAbajo, s1 := wire#w1)
      S_Coil( #EstadoMAQ.Error_MAQx )
   END_RUNG
   RUNG wire#powerrail
      I_Contact( #EM_Down )
   END_RUNG wire#w1
   // the same network as SCL:
   IF #EstadoZona.Rearme_CBx THEN
       #EstadoMAQ.Err_SeguridadAbajo := FALSE;   // RS flip-flop
   END_IF;
   IF NOT #EM_Down THEN #EstadoMAQ.Err_SeguridadAbajo := TRUE; END_IF;
   IF #EstadoMAQ.Err_SeguridadAbajo THEN #EstadoMAQ.Error_MAQx := TRUE; END_IF;
END_REGION

REGION Network 75: ERROR - De Posicion en el Reset - Inicializa Garras y Centradores Abiertos
   RUNG wire#powerrail
      Contact( #EstadoZona.Rearme_CBx )
      S_RS(operand := #EstadoMAQ.Err_PosicionEnReset, s1 := wire#w2)
      S_Coil( #EstadoMAQ.Error_MAQx )
   END_RUNG
   RUNG wire#powerrail
      Contact( #Reset_ET00 )
      wire#w1
      I_Contact( #CentradoresAbiertos )
   END_RUNG wire#w2
   RUNG wire#powerrail
      Contact( #Reset_ET01 )
   END_RUNG wire#w1
   RUNG wire#w1
      I_Contact( #GarrasAbiertas )
   END_RUNG wire#w2
   // the same network as SCL:
   IF #EstadoZona.Rearme_CBx THEN
       #EstadoMAQ.Err_PosicionEnReset := FALSE;   // RS flip-flop
   END_IF;
   IF (#Reset_ET00 OR #Reset_ET01) AND (NOT #CentradoresAbiertos OR NOT #GarrasAbiertas) THEN
       #EstadoMAQ.Err_PosicionEnReset := TRUE;
   END_IF;
   IF #EstadoMAQ.Err_PosicionEnReset THEN #EstadoMAQ.Error_MAQx := TRUE; END_IF;
END_REGION

REGION Network 76: TMP - ERROR - TimeOut de Elevacion
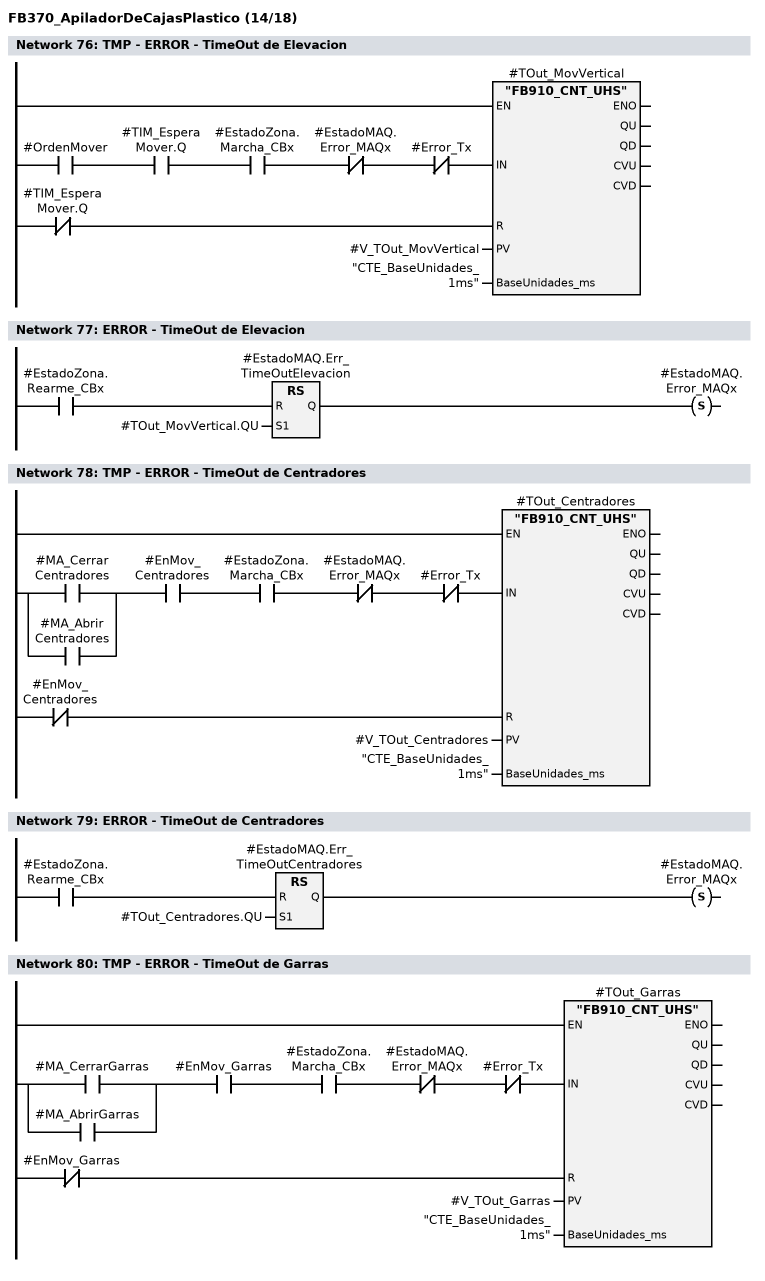
   RUNG wire#powerrail
      #TOut_MovVertical(IN := wire#w1, R := wire#w2, PV := #V_TOut_MovVertical, BaseUnidades_ms := "CTE_BaseUnidades_1ms", QU =>, QD =>, CVU =>, CVD =>)
   END_RUNG
   RUNG wire#powerrail
      Contact( #OrdenMover )
      Contact( #TIM_EsperaMover.Q )
      Contact( #EstadoZona.Marcha_CBx )
      I_Contact( #EstadoMAQ.Error_MAQx )
      I_Contact( #Error_Tx )
   END_RUNG wire#w1
   RUNG wire#powerrail
      I_Contact( #TIM_EsperaMover.Q )
   END_RUNG wire#w2
   // the same network as SCL:
   #TOut_MovVertical(IN := #OrdenMover AND #TIM_EsperaMover.Q AND #EstadoZona.Marcha_CBx AND NOT #EstadoMAQ.Error_MAQx AND NOT #Error_Tx,   // "FB910_CNT_UHS"
                     R := NOT #TIM_EsperaMover.Q,
                     PV := #V_TOut_MovVertical,
                     BaseUnidades_ms := "CTE_BaseUnidades_1ms");
END_REGION

REGION Network 77: ERROR - TimeOut de Elevacion
   RUNG wire#powerrail
      Contact( #EstadoZona.Rearme_CBx )
      S_RS(operand := #EstadoMAQ.Err_TimeOutElevacion, s1 := #TOut_MovVertical.QU)
      S_Coil( #EstadoMAQ.Error_MAQx )
   END_RUNG
   // the same network as SCL:
   IF #EstadoZona.Rearme_CBx THEN
       #EstadoMAQ.Err_TimeOutElevacion := FALSE;   // RS flip-flop
   END_IF;
   IF #TOut_MovVertical.QU THEN #EstadoMAQ.Err_TimeOutElevacion := TRUE; END_IF;
   IF #EstadoMAQ.Err_TimeOutElevacion THEN #EstadoMAQ.Error_MAQx := TRUE; END_IF;
END_REGION

REGION Network 78: TMP - ERROR - TimeOut de Centradores
   RUNG wire#powerrail
      #TOut_Centradores(IN := wire#w2, R := wire#w3, PV := #V_TOut_Centradores, BaseUnidades_ms := "CTE_BaseUnidades_1ms", QU =>, QD =>, CVU =>, CVD =>)
   END_RUNG
   RUNG wire#powerrail
      Contact( #MA_CerrarCentradores )
      wire#w1
      Contact( #EnMov_Centradores )
      Contact( #EstadoZona.Marcha_CBx )
      I_Contact( #EstadoMAQ.Error_MAQx )
      I_Contact( #Error_Tx )
   END_RUNG wire#w2
   RUNG wire#powerrail
      Contact( #MA_AbrirCentradores )
   END_RUNG wire#w1
   RUNG wire#powerrail
      I_Contact( #EnMov_Centradores )
   END_RUNG wire#w3
   // the same network as SCL:
   #TOut_Centradores(IN := (#MA_CerrarCentradores OR #MA_AbrirCentradores) AND #EnMov_Centradores AND #EstadoZona.Marcha_CBx AND NOT #EstadoMAQ.Error_MAQx AND NOT #Error_Tx,   // "FB910_CNT_UHS"
                     R := NOT #EnMov_Centradores,
                     PV := #V_TOut_Centradores,
                     BaseUnidades_ms := "CTE_BaseUnidades_1ms");
END_REGION

REGION Network 79: ERROR - TimeOut de Centradores
   RUNG wire#powerrail
      Contact( #EstadoZona.Rearme_CBx )
      S_RS(operand := #EstadoMAQ.Err_TimeOutCentradores, s1 := #TOut_Centradores.QU)
      S_Coil( #EstadoMAQ.Error_MAQx )
   END_RUNG
   // the same network as SCL:
   IF #EstadoZona.Rearme_CBx THEN
       #EstadoMAQ.Err_TimeOutCentradores := FALSE;   // RS flip-flop
   END_IF;
   IF #TOut_Centradores.QU THEN #EstadoMAQ.Err_TimeOutCentradores := TRUE; END_IF;
   IF #EstadoMAQ.Err_TimeOutCentradores THEN #EstadoMAQ.Error_MAQx := TRUE; END_IF;
END_REGION

REGION Network 80: TMP - ERROR - TimeOut de Garras
   RUNG wire#powerrail
      #TOut_Garras(IN := wire#w2, R := wire#w3, PV := #V_TOut_Garras, BaseUnidades_ms := "CTE_BaseUnidades_1ms", QU =>, QD =>, CVU =>, CVD =>)
   END_RUNG
   RUNG wire#powerrail
      Contact( #MA_CerrarGarras )
      wire#w1
      Contact( #EnMov_Garras )
      Contact( #EstadoZona.Marcha_CBx )
      I_Contact( #EstadoMAQ.Error_MAQx )
      I_Contact( #Error_Tx )
   END_RUNG wire#w2
   RUNG wire#powerrail
      Contact( #MA_AbrirGarras )
   END_RUNG wire#w1
   RUNG wire#powerrail
      I_Contact( #EnMov_Garras )
   END_RUNG wire#w3
   // the same network as SCL:
   #TOut_Garras(IN := (#MA_CerrarGarras OR #MA_AbrirGarras) AND #EnMov_Garras AND #EstadoZona.Marcha_CBx AND NOT #EstadoMAQ.Error_MAQx AND NOT #Error_Tx,   // "FB910_CNT_UHS"
                R := NOT #EnMov_Garras,
                PV := #V_TOut_Garras,
                BaseUnidades_ms := "CTE_BaseUnidades_1ms");
END_REGION

REGION Network 81: ERROR - TimeOut de Garras
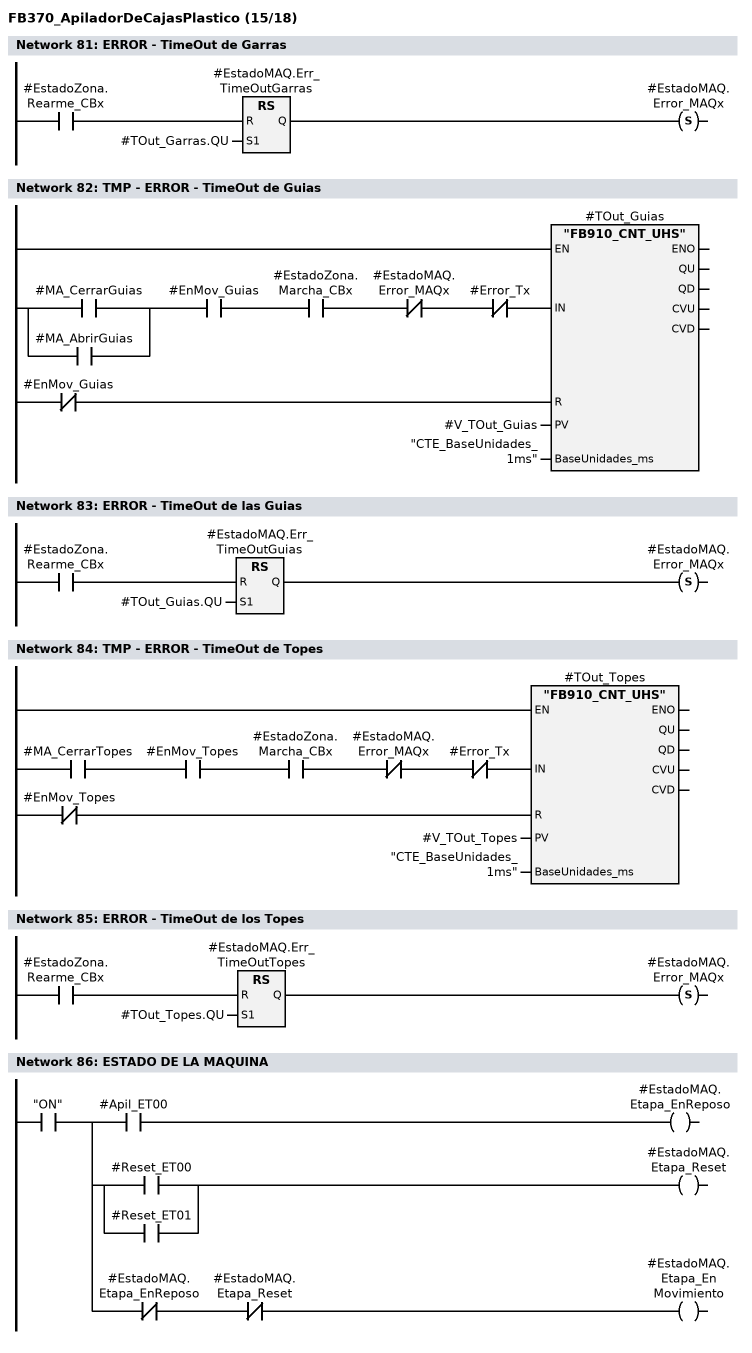
   RUNG wire#powerrail
      Contact( #EstadoZona.Rearme_CBx )
      S_RS(operand := #EstadoMAQ.Err_TimeOutGarras, s1 := #TOut_Garras.QU)
      S_Coil( #EstadoMAQ.Error_MAQx )
   END_RUNG
   // the same network as SCL:
   IF #EstadoZona.Rearme_CBx THEN
       #EstadoMAQ.Err_TimeOutGarras := FALSE;   // RS flip-flop
   END_IF;
   IF #TOut_Garras.QU THEN #EstadoMAQ.Err_TimeOutGarras := TRUE; END_IF;
   IF #EstadoMAQ.Err_TimeOutGarras THEN #EstadoMAQ.Error_MAQx := TRUE; END_IF;
END_REGION

REGION Network 82: TMP - ERROR - TimeOut de Guias
   RUNG wire#powerrail
      #TOut_Guias(IN := wire#w2, R := wire#w3, PV := #V_TOut_Guias, BaseUnidades_ms := "CTE_BaseUnidades_1ms", QU =>, QD =>, CVU =>, CVD =>)
   END_RUNG
   RUNG wire#powerrail
      Contact( #MA_CerrarGuias )
      wire#w1
      Contact( #EnMov_Guias )
      Contact( #EstadoZona.Marcha_CBx )
      I_Contact( #EstadoMAQ.Error_MAQx )
      I_Contact( #Error_Tx )
   END_RUNG wire#w2
   RUNG wire#powerrail
      Contact( #MA_AbrirGuias )
   END_RUNG wire#w1
   RUNG wire#powerrail
      I_Contact( #EnMov_Guias )
   END_RUNG wire#w3
   // the same network as SCL:
   #TOut_Guias(IN := (#MA_CerrarGuias OR #MA_AbrirGuias) AND #EnMov_Guias AND #EstadoZona.Marcha_CBx AND NOT #EstadoMAQ.Error_MAQx AND NOT #Error_Tx,   // "FB910_CNT_UHS"
               R := NOT #EnMov_Guias,
               PV := #V_TOut_Guias,
               BaseUnidades_ms := "CTE_BaseUnidades_1ms");
END_REGION

REGION Network 83: ERROR - TimeOut de las Guias
   RUNG wire#powerrail
      Contact( #EstadoZona.Rearme_CBx )
      S_RS(operand := #EstadoMAQ.Err_TimeOutGuias, s1 := #TOut_Guias.QU)
      S_Coil( #EstadoMAQ.Error_MAQx )
   END_RUNG
   // the same network as SCL:
   IF #EstadoZona.Rearme_CBx THEN
       #EstadoMAQ.Err_TimeOutGuias := FALSE;   // RS flip-flop
   END_IF;
   IF #TOut_Guias.QU THEN #EstadoMAQ.Err_TimeOutGuias := TRUE; END_IF;
   IF #EstadoMAQ.Err_TimeOutGuias THEN #EstadoMAQ.Error_MAQx := TRUE; END_IF;
END_REGION

REGION Network 84: TMP - ERROR - TimeOut de Topes
   RUNG wire#powerrail
      #TOut_Topes(IN := wire#w1, R := wire#w2, PV := #V_TOut_Topes, BaseUnidades_ms := "CTE_BaseUnidades_1ms", QU =>, QD =>, CVU =>, CVD =>)
   END_RUNG
   RUNG wire#powerrail
      Contact( #MA_CerrarTopes )
      Contact( #EnMov_Topes )
      Contact( #EstadoZona.Marcha_CBx )
      I_Contact( #EstadoMAQ.Error_MAQx )
      I_Contact( #Error_Tx )
   END_RUNG wire#w1
   RUNG wire#powerrail
      I_Contact( #EnMov_Topes )
   END_RUNG wire#w2
   // the same network as SCL:
   #TOut_Topes(IN := #MA_CerrarTopes AND #EnMov_Topes AND #EstadoZona.Marcha_CBx AND NOT #EstadoMAQ.Error_MAQx AND NOT #Error_Tx,   // "FB910_CNT_UHS"
               R := NOT #EnMov_Topes,
               PV := #V_TOut_Topes,
               BaseUnidades_ms := "CTE_BaseUnidades_1ms");
END_REGION

REGION Network 85: ERROR - TimeOut de los Topes
   RUNG wire#powerrail
      Contact( #EstadoZona.Rearme_CBx )
      S_RS(operand := #EstadoMAQ.Err_TimeOutTopes, s1 := #TOut_Topes.QU)
      S_Coil( #EstadoMAQ.Error_MAQx )
   END_RUNG
   // the same network as SCL:
   IF #EstadoZona.Rearme_CBx THEN
       #EstadoMAQ.Err_TimeOutTopes := FALSE;   // RS flip-flop
   END_IF;
   IF #TOut_Topes.QU THEN #EstadoMAQ.Err_TimeOutTopes := TRUE; END_IF;
   IF #EstadoMAQ.Err_TimeOutTopes THEN #EstadoMAQ.Error_MAQx := TRUE; END_IF;
END_REGION

REGION Network 86: ESTADO DE LA MAQUINA
   RUNG wire#powerrail
      Contact( "ON" )
      wire#w1
      Contact( #Apil_ET00 )
      Coil( #EstadoMAQ.Etapa_EnReposo )
   END_RUNG
   RUNG wire#w1
      Contact( #Reset_ET00 )
      wire#w2
      Coil( #EstadoMAQ.Etapa_Reset )
   END_RUNG
   RUNG wire#w1
      Contact( #Reset_ET01 )
   END_RUNG wire#w2
   RUNG wire#w1
      I_Contact( #EstadoMAQ.Etapa_EnReposo )
      I_Contact( #EstadoMAQ.Etapa_Reset )
      Coil( #EstadoMAQ.Etapa_EnMovimiento )
   END_RUNG
   // the same network as SCL:
   #EstadoMAQ.Etapa_EnReposo := "ON" AND #Apil_ET00;
   #EstadoMAQ.Etapa_Reset := "ON" AND (#Reset_ET00 OR #Reset_ET01);
   #EstadoMAQ.Etapa_EnMovimiento := "ON" AND NOT #EstadoMAQ.Etapa_EnReposo AND NOT #EstadoMAQ.Etapa_Reset;
END_REGION

REGION Network 87: ---
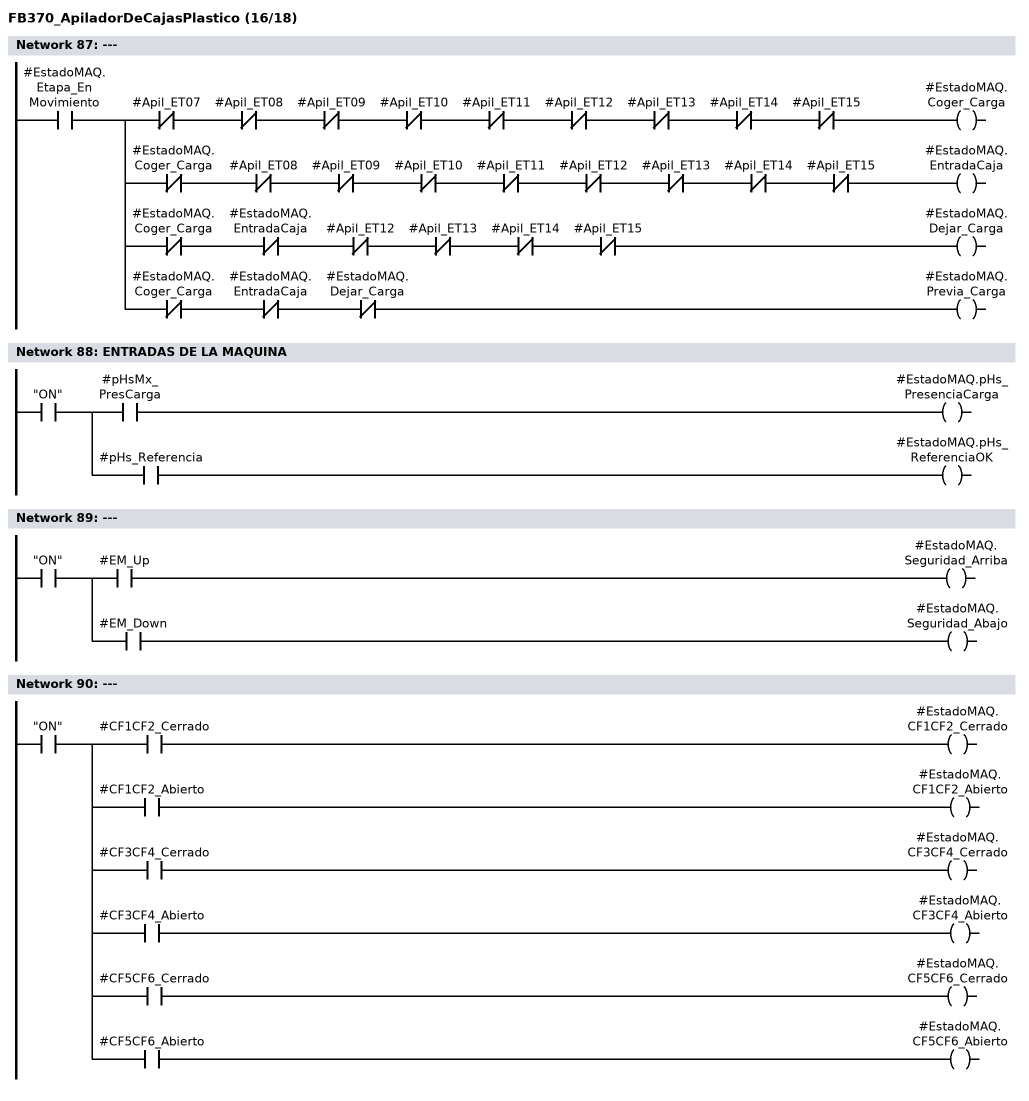
   RUNG wire#powerrail
      Contact( #EstadoMAQ.Etapa_EnMovimiento )
      wire#w1
      I_Contact( #Apil_ET07 )
      I_Contact( #Apil_ET08 )
      I_Contact( #Apil_ET09 )
      I_Contact( #Apil_ET10 )
      I_Contact( #Apil_ET11 )
      I_Contact( #Apil_ET12 )
      I_Contact( #Apil_ET13 )
      I_Contact( #Apil_ET14 )
      I_Contact( #Apil_ET15 )
      Coil( #EstadoMAQ.Coger_Carga )
   END_RUNG
   RUNG wire#w1
      I_Contact( #EstadoMAQ.Coger_Carga )
      I_Contact( #Apil_ET08 )
      I_Contact( #Apil_ET09 )
      I_Contact( #Apil_ET10 )
      I_Contact( #Apil_ET11 )
      I_Contact( #Apil_ET12 )
      I_Contact( #Apil_ET13 )
      I_Contact( #Apil_ET14 )
      I_Contact( #Apil_ET15 )
      Coil( #EstadoMAQ.EntradaCaja )
   END_RUNG
   RUNG wire#w1
      I_Contact( #EstadoMAQ.Coger_Carga )
      I_Contact( #EstadoMAQ.EntradaCaja )
      I_Contact( #Apil_ET12 )
      I_Contact( #Apil_ET13 )
      I_Contact( #Apil_ET14 )
      I_Contact( #Apil_ET15 )
      Coil( #EstadoMAQ.Dejar_Carga )
   END_RUNG
   RUNG wire#w1
      I_Contact( #EstadoMAQ.Coger_Carga )
      I_Contact( #EstadoMAQ.EntradaCaja )
      I_Contact( #EstadoMAQ.Dejar_Carga )
      Coil( #EstadoMAQ.Previa_Carga )
   END_RUNG
   // the same network as SCL:
   #EstadoMAQ.Coger_Carga := #EstadoMAQ.Etapa_EnMovimiento AND NOT #Apil_ET07 AND NOT #Apil_ET08 AND NOT #Apil_ET09 AND NOT #Apil_ET10 AND NOT #Apil_ET11 AND NOT #Apil_ET12 AND NOT #Apil_ET13 AND NOT #Apil_ET14 AND NOT #Apil_ET15;
   #EstadoMAQ.EntradaCaja := #EstadoMAQ.Etapa_EnMovimiento AND NOT #EstadoMAQ.Coger_Carga AND NOT #Apil_ET08 AND NOT #Apil_ET09 AND NOT #Apil_ET10 AND NOT #Apil_ET11 AND NOT #Apil_ET12 AND NOT #Apil_ET13 AND NOT #Apil_ET14 AND NOT #Apil_ET15;
   #EstadoMAQ.Dejar_Carga := #EstadoMAQ.Etapa_EnMovimiento AND NOT #EstadoMAQ.Coger_Carga AND NOT #EstadoMAQ.EntradaCaja AND NOT #Apil_ET12 AND NOT #Apil_ET13 AND NOT #Apil_ET14 AND NOT #Apil_ET15;
   #EstadoMAQ.Previa_Carga := #EstadoMAQ.Etapa_EnMovimiento AND NOT #EstadoMAQ.Coger_Carga AND NOT #EstadoMAQ.EntradaCaja AND NOT #EstadoMAQ.Dejar_Carga;
END_REGION

REGION Network 88: ENTRADAS DE LA MAQUINA
   RUNG wire#powerrail
      Contact( "ON" )
      wire#w1
      Contact( #pHsMx_PresCarga )
      Coil( #EstadoMAQ.pHs_PresenciaCarga )
   END_RUNG
   RUNG wire#w1
      Contact( #pHs_Referencia )
      Coil( #EstadoMAQ.pHs_ReferenciaOK )
   END_RUNG
   // the same network as SCL:
   #EstadoMAQ.pHs_PresenciaCarga := "ON" AND #pHsMx_PresCarga;
   #EstadoMAQ.pHs_ReferenciaOK := "ON" AND #pHs_Referencia;
END_REGION

REGION Network 89: ---
   RUNG wire#powerrail
      Contact( "ON" )
      wire#w1
      Contact( #EM_Up )
      Coil( #EstadoMAQ.Seguridad_Arriba )
   END_RUNG
   RUNG wire#w1
      Contact( #EM_Down )
      Coil( #EstadoMAQ.Seguridad_Abajo )
   END_RUNG
   // the same network as SCL:
   #EstadoMAQ.Seguridad_Arriba := "ON" AND #EM_Up;
   #EstadoMAQ.Seguridad_Abajo := "ON" AND #EM_Down;
END_REGION

REGION Network 90: ---
   RUNG wire#powerrail
      Contact( "ON" )
      wire#w1
      Contact( #CF1CF2_Cerrado )
      Coil( #EstadoMAQ.CF1CF2_Cerrado )
   END_RUNG
   RUNG wire#w1
      Contact( #CF1CF2_Abierto )
      Coil( #EstadoMAQ.CF1CF2_Abierto )
   END_RUNG
   RUNG wire#w1
      Contact( #CF3CF4_Cerrado )
      Coil( #EstadoMAQ.CF3CF4_Cerrado )
   END_RUNG
   RUNG wire#w1
      Contact( #CF3CF4_Abierto )
      Coil( #EstadoMAQ.CF3CF4_Abierto )
   END_RUNG
   RUNG wire#w1
      Contact( #CF5CF6_Cerrado )
      Coil( #EstadoMAQ.CF5CF6_Cerrado )
   END_RUNG
   RUNG wire#w1
      Contact( #CF5CF6_Abierto )
      Coil( #EstadoMAQ.CF5CF6_Abierto )
   END_RUNG
   // the same network as SCL:
   #EstadoMAQ.CF1CF2_Cerrado := "ON" AND #CF1CF2_Cerrado;
   #EstadoMAQ.CF1CF2_Abierto := "ON" AND #CF1CF2_Abierto;
   #EstadoMAQ.CF3CF4_Cerrado := "ON" AND #CF3CF4_Cerrado;
   #EstadoMAQ.CF3CF4_Abierto := "ON" AND #CF3CF4_Abierto;
   #EstadoMAQ.CF5CF6_Cerrado := "ON" AND #CF5CF6_Cerrado;
   #EstadoMAQ.CF5CF6_Abierto := "ON" AND #CF5CF6_Abierto;
END_REGION

REGION Network 91: ---
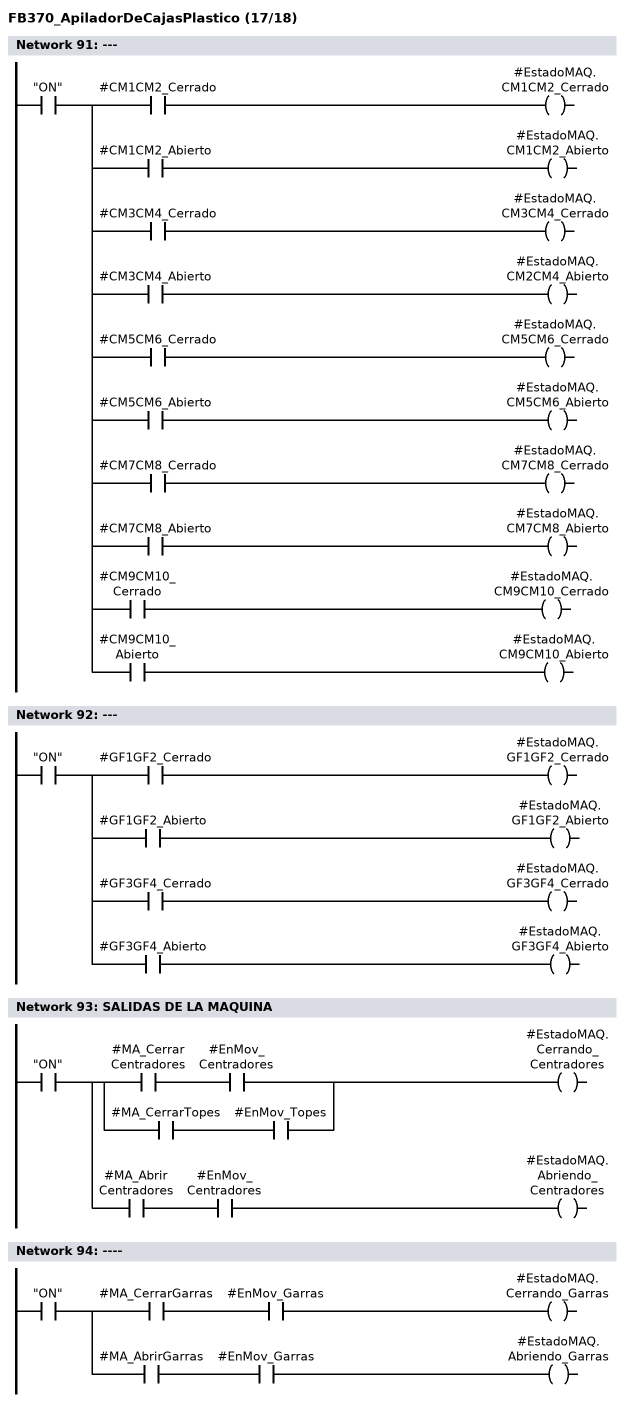
   RUNG wire#powerrail
      Contact( "ON" )
      wire#w1
      Contact( #CM1CM2_Cerrado )
      Coil( #EstadoMAQ.CM1CM2_Cerrado )
   END_RUNG
   RUNG wire#w1
      Contact( #CM1CM2_Abierto )
      Coil( #EstadoMAQ.CM1CM2_Abierto )
   END_RUNG
   RUNG wire#w1
      Contact( #CM3CM4_Cerrado )
      Coil( #EstadoMAQ.CM3CM4_Cerrado )
   END_RUNG
   RUNG wire#w1
      Contact( #CM3CM4_Abierto )
      Coil( #EstadoMAQ.CM2CM4_Abierto )
   END_RUNG
   RUNG wire#w1
      Contact( #CM5CM6_Cerrado )
      Coil( #EstadoMAQ.CM5CM6_Cerrado )
   END_RUNG
   RUNG wire#w1
      Contact( #CM5CM6_Abierto )
      Coil( #EstadoMAQ.CM5CM6_Abierto )
   END_RUNG
   RUNG wire#w1
      Contact( #CM7CM8_Cerrado )
      Coil( #EstadoMAQ.CM7CM8_Cerrado )
   END_RUNG
   RUNG wire#w1
      Contact( #CM7CM8_Abierto )
      Coil( #EstadoMAQ.CM7CM8_Abierto )
   END_RUNG
   RUNG wire#w1
      Contact( #CM9CM10_Cerrado )
      Coil( #EstadoMAQ.CM9CM10_Cerrado )
   END_RUNG
   RUNG wire#w1
      Contact( #CM9CM10_Abierto )
      Coil( #EstadoMAQ.CM9CM10_Abierto )
   END_RUNG
   // the same network as SCL:
   #EstadoMAQ.CM1CM2_Cerrado := "ON" AND #CM1CM2_Cerrado;
   #EstadoMAQ.CM1CM2_Abierto := "ON" AND #CM1CM2_Abierto;
   #EstadoMAQ.CM3CM4_Cerrado := "ON" AND #CM3CM4_Cerrado;
   #EstadoMAQ.CM2CM4_Abierto := "ON" AND #CM3CM4_Abierto;
   #EstadoMAQ.CM5CM6_Cerrado := "ON" AND #CM5CM6_Cerrado;
   #EstadoMAQ.CM5CM6_Abierto := "ON" AND #CM5CM6_Abierto;
   #EstadoMAQ.CM7CM8_Cerrado := "ON" AND #CM7CM8_Cerrado;
   #EstadoMAQ.CM7CM8_Abierto := "ON" AND #CM7CM8_Abierto;
   #EstadoMAQ.CM9CM10_Cerrado := "ON" AND #CM9CM10_Cerrado;
   #EstadoMAQ.CM9CM10_Abierto := "ON" AND #CM9CM10_Abierto;
END_REGION

REGION Network 92: ---
   RUNG wire#powerrail
      Contact( "ON" )
      wire#w1
      Contact( #GF1GF2_Cerrado )
      Coil( #EstadoMAQ.GF1GF2_Cerrado )
   END_RUNG
   RUNG wire#w1
      Contact( #GF1GF2_Abierto )
      Coil( #EstadoMAQ.GF1GF2_Abierto )
   END_RUNG
   RUNG wire#w1
      Contact( #GF3GF4_Cerrado )
      Coil( #EstadoMAQ.GF3GF4_Cerrado )
   END_RUNG
   RUNG wire#w1
      Contact( #GF3GF4_Abierto )
      Coil( #EstadoMAQ.GF3GF4_Abierto )
   END_RUNG
   // the same network as SCL:
   #EstadoMAQ.GF1GF2_Cerrado := "ON" AND #GF1GF2_Cerrado;
   #EstadoMAQ.GF1GF2_Abierto := "ON" AND #GF1GF2_Abierto;
   #EstadoMAQ.GF3GF4_Cerrado := "ON" AND #GF3GF4_Cerrado;
   #EstadoMAQ.GF3GF4_Abierto := "ON" AND #GF3GF4_Abierto;
END_REGION

REGION Network 93: SALIDAS DE LA MAQUINA
   RUNG wire#powerrail
      Contact( "ON" )
      wire#w1
      Contact( #MA_CerrarCentradores )
      Contact( #EnMov_Centradores )
      wire#w2
      Coil( #EstadoMAQ.Cerrando_Centradores )
   END_RUNG
   RUNG wire#w1
      Contact( #MA_CerrarTopes )
      Contact( #EnMov_Topes )
   END_RUNG wire#w2
   RUNG wire#w1
      Contact( #MA_AbrirCentradores )
      Contact( #EnMov_Centradores )
      Coil( #EstadoMAQ.Abriendo_Centradores )
   END_RUNG
   // the same network as SCL:
   #EstadoMAQ.Cerrando_Centradores := "ON" AND ((#MA_CerrarCentradores AND #EnMov_Centradores) OR (#MA_CerrarTopes AND #EnMov_Topes));
   #EstadoMAQ.Abriendo_Centradores := "ON" AND #MA_AbrirCentradores AND #EnMov_Centradores;
END_REGION

REGION Network 94: ----
   RUNG wire#powerrail
      Contact( "ON" )
      wire#w1
      Contact( #MA_CerrarGarras )
      Contact( #EnMov_Garras )
      Coil( #EstadoMAQ.Cerrando_Garras )
   END_RUNG
   RUNG wire#w1
      Contact( #MA_AbrirGarras )
      Contact( #EnMov_Garras )
      Coil( #EstadoMAQ.Abriendo_Garras )
   END_RUNG
   // the same network as SCL:
   #EstadoMAQ.Cerrando_Garras := "ON" AND #MA_CerrarGarras AND #EnMov_Garras;
   #EstadoMAQ.Abriendo_Garras := "ON" AND #MA_AbrirGarras AND #EnMov_Garras;
END_REGION

REGION Network 95: ----
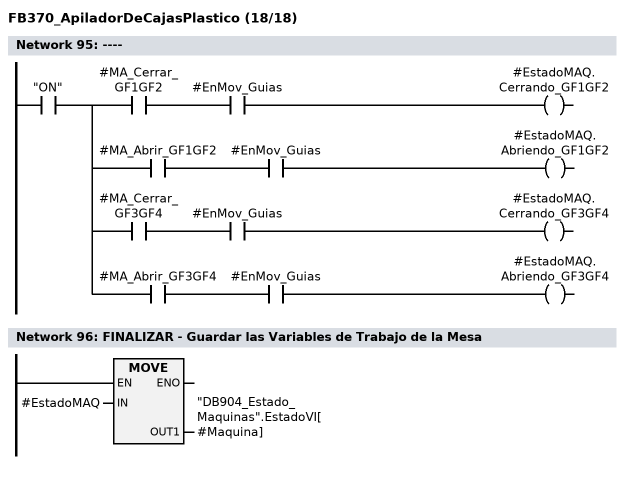
   RUNG wire#powerrail
      Contact( "ON" )
      wire#w1
      Contact( #MA_Cerrar_GF1GF2 )
      Contact( #EnMov_Guias )
      Coil( #EstadoMAQ.Cerrando_GF1GF2 )
   END_RUNG
   RUNG wire#w1
      Contact( #MA_Abrir_GF1GF2 )
      Contact( #EnMov_Guias )
      Coil( #EstadoMAQ.Abriendo_GF1GF2 )
   END_RUNG
   RUNG wire#w1
      Contact( #MA_Cerrar_GF3GF4 )
      Contact( #EnMov_Guias )
      Coil( #EstadoMAQ.Cerrando_GF3GF4 )
   END_RUNG
   RUNG wire#w1
      Contact( #MA_Abrir_GF3GF4 )
      Contact( #EnMov_Guias )
      Coil( #EstadoMAQ.Abriendo_GF3GF4 )
   END_RUNG
   // the same network as SCL:
   #EstadoMAQ.Cerrando_GF1GF2 := "ON" AND #MA_Cerrar_GF1GF2 AND #EnMov_Guias;
   #EstadoMAQ.Abriendo_GF1GF2 := "ON" AND #MA_Abrir_GF1GF2 AND #EnMov_Guias;
   #EstadoMAQ.Cerrando_GF3GF4 := "ON" AND #MA_Cerrar_GF3GF4 AND #EnMov_Guias;
   #EstadoMAQ.Abriendo_GF3GF4 := "ON" AND #MA_Abrir_GF3GF4 AND #EnMov_Guias;
END_REGION

REGION Network 96: FINALIZAR - Guardar las Variables de Trabajo de la Mesa
   RUNG wire#powerrail
      Move(in := #EstadoMAQ, out1 => "DB904_Estado_Maquinas".EstadoVI[#Maquina])
   END_RUNG
   // the same network as SCL:
   "DB904_Estado_Maquinas".EstadoVI[#Maquina] := #EstadoMAQ;
END_REGION
END_FUNCTION_BLOCK
